// TwinCAT 3 PLC project L2SIVacuum
// Title: LCLS Vacuum
// Company: SLAC - LCLS
// Author: LCLS ECS-Platforms
// ProjectVersion: 2.6.6
// ProgramVersion: 3.1.4026.17
// libraries:
//   LCLS General, * (SLAC)
//   PMPS, * (SLAC - LCLS)
//   Tc2_DataExchange, * (Beckhoff Automation GmbH)
//   Tc2_EtherCAT, * (Beckhoff Automation GmbH)
//   Tc2_ModbusSrv, * (Beckhoff Automation GmbH)
//   Tc2_SerialCom, * (Beckhoff Automation GmbH)
//   Tc2_Standard, * (Beckhoff Automation GmbH)
//   Tc2_System, * (Beckhoff Automation GmbH)
//   Tc2_TcpIp, * (Beckhoff Automation GmbH)
//   Tc2_Utilities, * (Beckhoff Automation GmbH)
//   Tc3_EventLogger, * (Beckhoff Automation GmbH)
//   Tc3_JsonXml, * (Beckhoff Automation GmbH)
//   Tc3_Module, * (Beckhoff Automation GmbH)
//   TcUnit, * (www.tcunit.org)
// project tree:
//   DUTs/Gauges/ E_PressureState.TcDUT, Gauge_Type.TcDUT, ST_VG.TcDUT
//   DUTs/LVDT/ ST_SerLVC4000.TcDUT
//   DUTs/Oerlikon/ ST_TD20Status.TcDUT, ST_TD400Control.TcDUT, ST_TD400Status.TcDUT
//   DUTs/Pfeiffer/ ST_PfeifferControl.TcDUT, ST_PfeifferStatus.TcDUT
//   DUTs/Pumps/ E_PumpState.TcDUT, ST_AgilentPTM.TcDUT, ST_EbaraDryPump.TcDUT, ST_EbaraEVA.TcDUT, ST_EbaraPTM.TcDUT, ST_KashiyamaDryPump.TcDUT, ST_LeyboldPTM.TcDUT, ST_PfeifferPTM.TcDUT, ST_PIP.TcDUT, ST_PTM.TcDUT, ST_RoughPump.TcDUT
//   DUTs/Valves/ E_ValvePositionState.TcDUT, E_VCN.TcDUT, E_2OO3_MODE.TcDUT, E_VGC.TcDUT, ST_ValveBase.TcDUT, ST_VFS.TcDUT, ST_VGC_2S.TcDUT, ST_VRC_NO.TcDUT, ST_VWC_NO.TcDUT, ST_VVC.TcDUT, ST_VCC_NO.TcDUT, ST_VCN.TcDUT, ST_VGC.TcDUT, ST_VRC.TcDUT
//   DUTs/Valves/VAT590/EtherCAT Interface/ E_ControlMode.TcDUT, E_ControlModeSP.TcDUT, E_FatalErrors.TcDUT, ST_ExtendedWarnings.TcDUT, ST_GeneralControlSP.TcDUT, ST_GeneralStatus.TcDUT, ST_GeneralWarnings.TcDUT
//   DUTs/Valves/VAT590/ E_VAT590_AccessMode.TcDUT, E_VAT590_PID_CTRL.TcDUT, E_VCN_VAT590.TcDUT, ST_CoEIndSub.TcDUT, ST_VAT590_COE.TcDUT, ST_VAT590_STATUS.TcDUT, ST_VCN_VAT590.TcDUT
//   GVLs/ Constants.TcGVL, Global_Variables.TcGVL, GVL_MacroSensorsParameters.TcGVL, GVL_PfeifferParameters.TcGVL
//   / PlcTask.TcTTO
//   POUs/ADS/ FB_ADS.TcPOU, FB_ADS_WATCHDOG.TcPOU, FB_TBOOL_ADS.TcPOU
//   POUs/Functions/Deprecated/Gauges/ FB_MKS317A.TcPOU, FB_MKS500_EP.TcPOU, FB_PressureState.TcPOU
//   POUs/Functions/Deprecated/Valves/ FB_VCC.TcPOU, FB_VCC_NO.TcPOU, FB_VGC_AP.TcPOU, FB_VGC_EBD.TcPOU
//   POUs/Functions/Gauges/ FB_901_ECAT.TcPOU, FB_9XX.TcPOU, FB_972.TcPOU, FB_IE514.TcPOU, FB_MX7M.TcPOU, FB_MKS355.TcPOU, FB_GaugeBase.TcPOU, FB_CVM201.TcPOU, FB_CCM501.TcPOU, FB_IMG401.TcPOU, FB_MKS909.TcPOU, FB_MKS909_RBK.TcPOU, FB_CMR362.TcPOU, FB_GCM.TcPOU, FB_ITR90.TcPOU, FB_MKS392.TcPOU, FB_MKS500.TcPOU, FB_MKS722.TcPOU, FB_MKS_937A.TcPOU, FB_MKS317.TcPOU, FB_MKS275.TcPOU, FB_MKS_937B.TcPOU, FB_MKS422.TcPOU
//   POUs/Functions/Gauges/Interfaces/ FB_GaugeModbus.TcPOU, FB_Gauge_Interface.TcPOU, FB_TGCC_ADS.TcPOU, FB_TGPI_ADS.TcPOU, FB_GaugeSelection.TcPOU (not stored)
//   POUs/Functions/Pumps/ FB_EbaraDryPump.TcPOU, FB_EbaraEVA.TcPOU, FB_KashiyamaPump.TcPOU, FB_KashiyamaPump_G.TcPOU, FB_PIP_Gamma.TcPOU, FB_PIP_Gamma_V2.TcPOU, FB_PIP_SIP.TcPOU, FB_PTM_Agilent.TcPOU, FB_PTM_Ebara_011M.TcPOU, FB_PTM_Ebara_010M.TcPOU, FB_PTM_MagDriveDigital.TcPOU, FB_PTM_Pfeiffer.TcPOU, FB_PTM_TurboDrive.TcPOU, FB_PTM_TwisTorr.TcPOU, FB_Pump.TcPOU, FB_ScrollPump.TcPOU
//   POUs/Functions/Pumps/functions/ FB_TurboExtLogic.TcPOU, F_TurboExtILK_NO.TcPOU, F_TurboExtILKLogic.TcPOU, F_TurboExtILKLogic_2.TcPOU, F_TurboExtILK_NO_1.TcPOU
//   POUs/Functions/Pumps/Interfaces/ FB_PIP_Interface_In.TcPOU, FB_PIP_Interface_Out.TcPOU, FB_TPIP_ADS.TcPOU
//   POUs/Functions/Valves/ FB_Kashiyama_VRC.TcPOU, FB_MKS248.TcPOU, FB_TurbVentvalve_NO.TcPOU, FB_Valve.TcPOU, FB_VCN_VAT590.TcPOU, FB_VFS.TcPOU, FB_VFS_2OO3.TcPOU, FB_VGC_2S.TcPOU, FB_VRC_DA.TcPOU, FB_VRC_EBD.TcPOU, FB_VRC_NC_ClsLS.TcPOU, FB_VRC_NO.TcPOU, FB_VRC_NO_FFO.TcPOU, FB_VVC.TcPOU, FB_VCN.TcPOU, FB_VGC.TcPOU, FB_VRC.TcPOU, FB_VRC_OK_CLS.TcPOU
//   POUs/Functions/Valves/functions/ F_RoughPumpInlet_ILK.TcPOU, F_TurboGateValve_ILK.TcPOU, F_TurboGateValve_ILK_1.TcPOU, F_TurboGateValve_Protection_ILK.TcPOU, F_TURBO_VRC_ILK.TcPOU, F_VALVE_REL_ILK.TcPOU, F_VRC_DIODE_ILK_OK.TcPOU, F_VRC_DIODE_ILK.TcPOU
//   POUs/Functions/Valves/Interfaces/ FB_TVGC_2S_ADS.TcPOU, FB_VFS_2OO3Interface.TcPOU, FB_VFS_Interface.TcPOU, FB_TVGC_ADS.TcPOU, FB_Valve_Interface.TcPOU, ITF_Valve.TcIO
//   POUs/Serial drivers/LVDT/MacroSensors/ FB_LVC4000Com.TcPOU, FB_LVC4000SerialDriver.TcPOU, FB_LVC4000Transaction.TcPOU
//   POUs/Serial drivers/Pumps/Oerlikon TD20/ FB_OERLIKON_TD20_COM.TcPOU, FB_OERLIKON_TO_PTM.TcPOU, FB_TD20SerialDriver.TcPOU, FB_TD20Transaction.TcPOU, F_CalcTD20Checksum.TcPOU
//   POUs/Serial drivers/Pumps/Oerlikon TD400/ FB_OERLIKON_TD400_COM.TcPOU, FB_OERLIKON_TD400_TO_PTM.TcPOU, FB_TD400SerialDriver.TcPOU, FB_TD400Transaction.TcPOU, F_CalcTD400Checksum.TcPOU
//   POUs/Serial drivers/Pumps/Pfeiffer/ FB_PfeifferSerialDriver.TcPOU, FB_PfeifferTransaction.TcPOU, FB_PFEIFFER_COM.TcPOU, FB_PFEIFFER_TO_PTM.TcPOU, F_CalcPfeifferCheckSum.TcPOU
//   UnitTests/Functions/ V_TO_INT.TcPOU
//   UnitTests/Gauges/ FB_GCC_Test.TcPOU, FB_GHC_Test.TcPOU, FB_GPI_Test.TcPOU
//   UnitTests/ PRG_Test.TcPOU
//   UnitTests/Pumps/ FB_PIP_Test.TcPOU, FB_PTM_Test.TcPOU
//   UnitTests/Valves/ FB_VGC_Test.TcPOU, FB_VRC_Test.TcPOU
//   Version/ Global_Version.TcGVL
// real-time tasks:
//   TASK TestTask: cycle T#10ms, priority 16, ADS port 350
// variable links:
//   L2SIVacuum/L2SIVacuum Instance <-> L2SIVacuum/L2SIVacuum Instance
//     PlcTask Inputs/PRG_Test.fb_GCC_Test.fb_MKS422.i_iPRESS_R <-> PlcTask Outputs/PRG_Test.fb_GCC_Test.i_iPRESS_R
//     PlcTask Inputs/PRG_Test.fb_GPI_Test.fb_MKS275.i_iPRESS_R <-> PlcTask Outputs/PRG_Test.fb_GPI_Test.i_iPRESS_R
//     PlcTask Inputs/PRG_Test.fb_GPI_Test.fb_MKS317.i_iPRESS_R <-> PlcTask Outputs/PRG_Test.fb_GPI_Test.i_iPRESS_R
//     PlcTask Inputs/PRG_Test.fb_PTM_Test.fb_PTM_Ebara_010M.i_iCurrentMon <-> PlcTask Outputs/PRG_Test.fb_PTM_Test.i_iCurrentMon
//     PlcTask Inputs/PRG_Test.fb_PTM_Test.fb_PTM_Ebara_010M.i_iRawSpeed <-> PlcTask Outputs/PRG_Test.fb_PTM_Test.i_iRawSpeed
//     PlcTask Inputs/PRG_Test.fb_PTM_Test.fb_PTM_Ebara_010M.i_iTempMon <-> PlcTask Outputs/PRG_Test.fb_PTM_Test.i_iTempMon
//     PlcTask Inputs/PRG_Test.fb_PTM_Test.q_iSpeedSet <-> PlcTask Outputs/PRG_Test.fb_PTM_Test.i_diCurSpd

CONFIGURATION L2SIVacuum
    RESOURCE PLC ON TwinCAT3
        TASK PlcTask(INTERVAL := T#10ms, PRIORITY := 16);
        PROGRAM PRG_Test WITH PlcTask : PRG_Test;
    END_RESOURCE
END_CONFIGURATION

// ---- DUTs/Gauges/E_PressureState.TcDUT
TYPE E_PressureState :
(
    // Invalid states
    Off,//	 //gc_GaugeValidState - 1,
    GaugeDisconnected, //gc_GaugeValidState -2,
    OoR, //gc_GaugeValidState -6,
    // Ion gauges
    PressInvalid, //gc_GaugeValidState - 3,
    Starting, //gc_GaugeValidState - 4

    //Valid States (Positive)
    Valid, // gc_GaugeValidState set in "Global Variable Folder: Constants"
    ValidHi, //gc_GaugeValidState + 1,
    ValidLo //gc_GaugeValidState + 2,

) INT;
END_TYPE

// ---- DUTs/Gauges/Gauge_Type.TcDUT
TYPE Gauge_Type: (
PG722B := 0, //Baraton Gauge
IG903 := 1 , //Cold Cathode
PG907 := 2 , //Pirani Gauge
IG909:= 3 , //Hot Cathode
PG925 := 4 ); //MicroPirani Gauge
(* This enumeration should match up with the EDM MUX button on the vacuum gauge expert controls screen *)
END_TYPE

// ---- DUTs/Gauges/ST_VG.TcDUT
TYPE ST_VG :
STRUCT
    /// A general gauge structure is used to make the rest of the interlocking simpler. There are some parameters for cold cathodes that are not used by pirani.
    ///These features aren't disabled, they just aren't used, think child/parent classes.
    ///
    {attribute 'pytmc' := '
    pv: PRESS;
    field: HOPR 1000
    field: LOPR 0
    field: PREC 2
    field: EGU "TORR"
    io: i;
    '}
    rPRESS: REAL;  //This is the human-readable pressure
    {attribute 'pytmc' := '
    pv: AT_VAC;
    io: i;
    field: ZNAM FALSE;
    field: ONAM TRUE;
    '}
    xAT_VAC: BOOL;
    {attribute 'pytmc' := '
    pv: PRESS_OK;
    field: ZNAM OFF;
    field: ONAM ON;
    io: i;
    '}
    xPRESS_OK: BOOL;
    {attribute 'pytmc' := '
    pv: STATE;
    field: ZRST Off;
    field: ONST GaugeDisconnected;
    field: TWST OoR;
    field: THST PressInvalid;
    field: FRST Starting;
    field: FVST Valid;
    field: SXST ValidHi;
    field: SVST ValidLo;
    io: i;
    '}
    eState	:	E_PressureState;
    (* EPICS Controls *)
    {attribute 'pytmc' := '
    pv: HV_SW;
    io: io;
    field: ZNAM OFF;
    field: ONAM ON;
    '}
    xHV_SW: BOOL; // High Voltage Switch from epics
    {attribute 'pytmc' := '
    pv: Auto_On;
    field: ZNAM FALSE;
    field: ONAM TRUE;
    io:io;
    '}
    xAutoOn : BOOL := TRUE;
    {attribute 'pytmc' := '
    pv: AutoOn_timer;
    io:i;
    '}
    iAutoOnTimer : INT;
    /// Controls and I/Os
    {attribute 'pytmc' := '
    pv: PRESS_AI;
    io: i;
    '}
    i_iPRESS_R  :INT; // input Pressure // Link to analog Input
    {attribute 'pytmc' := '
    pv: HV_ON;
    io: i;
    '}
    i_xHV_ON	: BOOL; //  True when High Voltage is on
    {attribute 'pytmc' := '
    pv: DISC_ACTIVE;
    field: ZNAM NO DISC;
    field: ONAM DISC ACTIVE;
    io: i;
    '}
    i_xDisc_Active : BOOL;// Discharge Current Active
    {attribute 'pytmc' := '
    pv: HV_DIS_DO;
    io: i;
    field: ZNAM FALSE ;
    field: ONAM TRUE ;
    '}
    q_xHV_DIS : BOOL; // Enable High Voltage when True
    //
    wHV_RO: WORD;

    /// Bakeout bit
    xBAKEOUT: BOOL;

    //enum for gauge type - will replace iType
    eTYPE: Gauge_Type := PG907;
    //Gauge type, deprecated (default to pirani)
    iTYPE: INT := 2;
    // Index location of the associated Pirani Gauge
    wPG: WORD;


    xTurnOnTime: BOOL;/// Turn on Timers for cold cathode warmup

    iVacSp	:	INT;/// At vacuum setpoint for all gauges
    {attribute 'pytmc' := '
    pv: VAC_SP;
    io:io;
    field: HOPR 1000
    field: LOPR 0
    field: PREC 2
    field: EGU "TORR"
    autosave_pass1: VAL DESC
    '}
    rVAC_SP: REAL := 0.001; /// At vacuum setpoint for all gauges
    /// Protection setpoint for ion gauges at which the gauge turns off, not used for pirani
    {attribute 'pytmc' := '
    pv: PRO_SP;
    io: io;
    field: HOPR 1000
    field: LOPR 0
    field: PREC 2
    field: EGU "TORR"
    autosave_pass1: VAL DESC
    '}
    rPRO_SP: REAL := 0.001;
    {attribute 'pytmc' := '
    pv: SP_HYS;
    io: io;
    field: HOPR 1000
    field: LOPR 0
    field: PREC 2
    field: EGU "TORR"
    autosave_pass1: VAL DESC
    '}
    /// Protection setpoint hysteresis
    rHYS_PR: REAL := 0.001;
    {attribute 'pytmc' := '
    pv: ILK_OK;
    field: ZNAM NOT OK ;
    field: ONAM OK ;
    io: i;
    '}
    xILKOk	:	BOOL; (* also a control *)
    {attribute 'pytmc' := '
    pv: LOGGER;
    io: io;
    field: ZNAM OFF ;
    field: ONAM ON ;
    '}
    xLog : BOOL:=TRUE;
    //Required for other devices using this gauge as interlock
    sPath: STRING;

    /// Full scale pressure in Torr for baratron pressure conversion
    rFULL_SCALE: REAL := 1000;

END_STRUCT
END_TYPE

// ---- DUTs/LVDT/ST_SerLVC4000.TcDUT
TYPE ST_SerLVC4000 :
STRUCT
    (* Readbacks *)
    {attribute 'pytmc' := '
    pv: voltage;
    io: i;
    '}
    i_iOut	:	INT; //Output voltage
    (* Controls *)
    {attribute 'pytmc' := '
    pv: ADC_COEFF;
    io: io;
    '}
    q_rADCsl	:	REAL; //ADC slope coeff
    {attribute 'pytmc' := '
    pv: ADC_OFFSET;
    io: io;
    '}
    q_rADCos	:	REAL; //ADC offset
    {attribute 'pytmc' := '
    pv: CALIB_SET;
    io: io;
    '}
    q_xCal	:	BOOL; //Activate calibration mode
    {attribute 'pytmc' := '
    pv: DISP_SET;
    io: io;
    '}
    q_xFull	:	BOOL; //Set full displacement during calibration
    {attribute 'pytmc' := '
    pv: ZERO_SET;
    io: io;
    '}
    q_xZero	:	BOOL; //Set zero during calibration
    {attribute 'pytmc' := '
    pv: GAIN_SET;
    io: io;
    '}
    q_iGain	:	INT; //Set instrument gain
    {attribute 'pytmc' := '
    pv: CALIB_ABORT;
    io: io;
    '}
    q_xAbortCal	:	BOOL; //Abort calibration mode
    (* Internal params *)
    {attribute 'pytmc' := '
    pv: ADDR;
    io: io;
    '}
    iAddr	:	INT; //RS485 address
    xTimeout	:	BOOL; //Timeout (true if no comm)
END_STRUCT
END_TYPE

// ---- DUTs/Oerlikon/ST_TD20Status.TcDUT
TYPE ST_TD20Status :  (* Serial communication defined in Oerlikon Leybold Manual 17200048 *)
STRUCT
    /// Received Status Word
    wStatusWord: WORD;
    /// Current stator frequency
    {attribute 'pytmc' := '
    pv: Frequency;
    io: i;
    '}
    wFrequency_P3: WORD;
    /// Current intermediate circuit voltage
    {attribute 'pytmc' := '
    pv: Voltage;
    io: i;
    '}
    wVoltage_P4: WORD;
    /// Current motor current
    {attribute 'pytmc' := '
    pv: MotorCurrent;
    io: i;
    '}
    wMotorCurrent_P5: WORD;
    /// Current frequency converter temperature
    {attribute 'pytmc' := '
    pv: Temperature;
    io: i;
    '}
    wConverterTemp_P11: WORD;
    /// Critical frequency
    {attribute 'pytmc' := '
    pv: CriticalFrequency;
    io: i;
    '}
    wCriticalFreq_P20: WORD;
    /// Max. Current Factor
    {attribute 'pytmc' := '
    pv: MaxCurrentFactor;
    io: i;
    '}
    wMaxCurrentFactor_P21: WORD;
    /// Setpoint Frequecy
    {attribute 'pytmc' := '
    pv: SetPointFreq;
    io: i;
    '}
    wSetpointFreq_P24: WORD;
    /// Max. run up time
    {attribute 'pytmc' := '
    pv: MaxRunUpTime;
    io: i;
    '}
    wMaxRunUpTime_P32: WORD;
    /// Current pump temperature
    {attribute 'pytmc' := '
    pv: PumpTemp;
    io: i;
    '}
    wPumpTemp_P127: WORD;
    /// most recent error code
    {attribute 'pytmc' := '
    pv: ErrorCode;
    io: i;
    '}
    wErrorCode_P171: WORD;
END_STRUCT
END_TYPE

// ---- DUTs/Oerlikon/ST_TD400Control.TcDUT
TYPE ST_TD400Control :  (* Serial communication defined in Oerlikon Leybold Manual GA05281_002_C0 *)
STRUCT
    {attribute 'pytmc' := '
    pv: SetPumpSpeed;
    io: i;
    '}
    wSetSetpointFreq_P24: WORD; // speed setting in Hz
END_STRUCT
END_TYPE

// ---- DUTs/Oerlikon/ST_TD400Status.TcDUT
TYPE ST_TD400Status :  (* Serial communication defined in Oerlikon Leybold Manual 17200048 *)
STRUCT
    /// Received Status Word
    wStatusWord: WORD;
    /// Current stator frequency
    {attribute 'pytmc' := '
    pv: Frequency;
    io: i;
    '}
    wFrequency_P3: WORD;
    /// Current intermediate circuit voltage
    {attribute 'pytmc' := '
    pv: Voltage;
    io: i;
    '}
    wVoltage_P4: WORD;
    /// Current motor current
    {attribute 'pytmc' := '
    pv: MotorCurrent;
    io: i;
    '}
    wMotorCurrent_P5: WORD;
    /// Current frequency converter temperature
    {attribute 'pytmc' := '
    pv: Temperature;
    io: i;
    '}
    wConverterTemp_P11: WORD;
    /// Maximum setpoint frequency
    {attribute 'pytmc' := '
    pv: MaxSetpoinFreq;
    io: i;
    '}
    wMaxSetpointFreq_P18: WORD;
    /// Minimum setpoint frequency
    {attribute 'pytmc' := '
    pv: MinSetpoinFreq;
    io: i;
    '}
    wMinSetpointFreq_P19: WORD;
    /// Critical frequency
    {attribute 'pytmc' := '
    pv: CriticalFrequency;
    io: i;
    '}
    wCriticalFreq_P20: WORD;
    /// Setpoint Frequecy
    {attribute 'pytmc' := '
    pv: SetPointFreq;
    io: i;
    '}
    wSetpointFreq_P24: WORD;
    /// Max. run up time
    {attribute 'pytmc' := '
    pv: MaxRunUpTime;
    io: i;
    '}
    wMaxRunUpTime_P32: WORD;
    /// Current pump temperature
    {attribute 'pytmc' := '
    pv: PumpTemp;
    io: i;
    '}
    wPumpTemp_P127: WORD;
    /// most recent error code
    {attribute 'pytmc' := '
    pv: ErrorCode;
    io: i;
    '}
    wErrorCode_P171: WORD;
END_STRUCT
END_TYPE

// ---- DUTs/Pfeiffer/ST_PfeifferControl.TcDUT
TYPE ST_PfeifferControl :
STRUCT
    /// enables communication
    {attribute 'pytmc' := '
    pv: COMM_EN;
    io: io;
    '}
    xEnableComm: BOOL;
    /// RS-485 Address
    {attribute 'pytmc' := '
    pv: ADDR;
    io: io;
    '}
    iSerialAddress: INT;
    {attribute 'pytmc' := '
    pv: EXT_ILK_OK;
    field: ZNAM ILK ACTIVE;
    field: ONAM ILK OK;
    io: i;
    '}
    /// pumping station (equivalent to ilk bit for varian)
    xPumpingStation_010: BOOL;
    {attribute 'pytmc' := '
    pv: SetPumpSpeed;
    io: i;
    '}
    iSetRotationSpeed_707: INT :=100; /// speed setting in % (normally 100%)
    /// RUN_DO bit
    {attribute 'pytmc' := '
    pv: RUN_DO;
    io: i;
    '}
    xMotorPump_023: BOOL;
    {attribute 'pytmc' := '
    pv: GAS_MODE;
    io: io;
    '}
    iGasMode_027: INT;
    /// interlock bit
     {attribute 'pytmc' := '
    pv: ILK_OK;
    field: ZNAM ILK ACTIVE;
    field: ONAM ILK OK;
    io: i;
    '}
    xIlk: BOOL;
    /// run/start bit
    {attribute 'pytmc' := '
    pv: RUN_SW;
    io: io;
    '}
    xRunSW: BOOL;
    /// error acknowledgement/reset bit
    {attribute 'pytmc' := '
    pv: ERR_RST;
    io: io;
    '}
    xErrorAck_009: BOOL;
    /// power consumption setting in % (normally 100%)
    uiPowerPct_708: UINT;
    xSetSpdMode_026: BOOL;
END_STRUCT
END_TYPE

// ---- DUTs/Pfeiffer/ST_PfeifferStatus.TcDUT
TYPE ST_PfeifferStatus :
STRUCT
    {attribute 'pytmc' := '
    pv: PumpingStation_RBV;
    field: ZNAM ILK ACTIVE;
    field: ONAM ILK OK;
    io: i;
    '}
    xPumpingStation_010: BOOL;
    {attribute 'pytmc' := '
    pv: PumpingStation_RBV;
    field: ZNAM FALSE;
    field: ONAM TRUE;
    io: i;
    '}
    xMotorPump_023: BOOL;
    {attribute 'pytmc' := '
    pv: GasMode_RBV;
    io: i;
    '}
    iGasMode_027: INT;
    {attribute 'pytmc' := '
    pv: ErrorMessage_RBV;
    io: i;
    '}
    sErrorCode_303: STRING;
    {attribute 'pytmc' := '
    pv: ErrorCode_RBV;
    io: i;
    '}
    iErrorCode_303	:	INT;
    {attribute 'pytmc' := '
    pv: WarningCode_RBV;
    io: i;
    '}
    iWarningCode_303	:	INT;
    {attribute 'pytmc' := '
    pv: ExcessPumpTemp_RBV;
    field: ZNAM FALSE;
    field: ONAM TRUE;
    io: i;
    '}
    xExcessTempPump_305: BOOL;
    {attribute 'pytmc' := '
    pv: TotationSpeedAttn_RBV;
    field: ZNAM FALSE;
    field: ONAM TRUE;
    io: i;
    '}
    xRotationSpeedAttn_306: BOOL;
    {attribute 'pytmc' := '
    pv: PumpAccelerating_RBV;
    field: ZNAM FALSE;
    field: ONAM TRUE;
    io: i;
    '}
    xPumpAccelerating_307: BOOL;
    {attribute 'pytmc' := '
    pv: PumpSpeed_RBV;
    io: i;
    '}
    diActiveRotationSpeed_309: DINT;
    {attribute 'pytmc' := '
    pv: DriveCurrent_RBV;
    io: i;
    '}
    lrDriveCurrent_310: LREAL;
    {attribute 'pytmc' := '
    pv: DrivePower_RBV;
    io: i;
    '}
    diDrivePower_316: DINT;
    {attribute 'pytmc' := '
    pv: TempElect_RBV;
    io: i;
    '}
    diTempElec_326: DINT;
    {attribute 'pytmc' := '
    pv: TempPump_RBV;
    io: i;
    '}
    diTempPmpBot_330: DINT;
    {attribute 'pytmc' := '
    pv: TempBearing_RBV;
    io: i;
    '}
    diTempBearng_342: DINT;
    {attribute 'pytmc' := '
    pv: TempMotor_RBV;
    io: i;
    '}
    diTempMotor_346: DINT;
    {attribute 'pytmc' := '
    pv: Power_RBV;
    io: i;
    '}
    uiPowerPct_708: UINT;
    {attribute 'pytmc' := '
    pv: Timeout_RBV;
    field: ZNAM FALSE;
    field: ONAM TRUE;
    io: i;
    '}
    xTimeout: BOOL;
    iSetRotationSpeed_707 : INT;
    iSetSpdMode_026: INT;
    xErrorAcknowledged: BOOL; //Not actually read back from the pump, but tells us ErrAck has processed
END_STRUCT
END_TYPE

// ---- DUTs/Pumps/E_PumpState.TcDUT
TYPE E_PumpState :
(
pumpSTOPPED	:= 0,
pumpSTARTING	:= 1,
pumpRUNNING	:= 2,
pumpFAULT := 3,
pumpSTOPPING :=4
);
END_TYPE

// ---- DUTs/Pumps/ST_AgilentPTM.TcDUT
TYPE ST_AgilentPTM EXTENDS ST_PTM :
STRUCT

(* Inputs *)
    (* 24V in Ramp state; 0V for others *)
    {attribute 'pytmc' := '
    pv: START;
    field: ZNAM FALSE;
    field: ONAM TRUE;
    io: i;
    '}
    i_xSTART :	BOOL;

    (* setpoint related to frequency *)
    {attribute 'pytmc' := '
    pv: R1Status;
    field: ZNAM FALSE;
    field: ONAM AT SPEED;
    io: i;
    '}
    i_xR1	:  BOOL;

    (* setpoint related to Power *)
    {attribute 'pytmc' := '
    pv: R2Status;
    field: ZNAM FALSE;
    field: ONAM TRUE;
    io: i;
    '}
    i_xR2	:  BOOL;

    (* low speed mode *)
    {attribute 'pytmc' := '
    pv: LSPD;
    field: ZNAM FALSE;
    field: ONAM TRUE;
    io: i;
    '}
    i_xLSpd	:  BOOL;


    (* Fault input*)
    //i_xFault : BOOL;  Inherit ST_PTM.xFault



(* controls *)
    (* Start/Stop -
        q_RunDo ;   Inherit ST_PTM.
     *)

    (* Low speed control *)
    {attribute 'pytmc' := '
    pv: LSPD_DO;
    field: ZNAM FALSE;
    field: ONAM TRUE;
    io: i;
    '}
    q_xLSpd		:  BOOL;

    (*Soft start *)
    {attribute 'pytmc' := '
    pv: XSS_DO;
    field: ZNAM FALSE;
    field: ONAM TRUE;
    io: i;
    '}
    q_xSS   	:  BOOL;

    (*pump Lock*)
    {attribute 'pytmc' := '
    pv: FaultLock;
    field: ZNAM FALSE;
    field: ONAM TRUE;
    io: i;
    '}
    xPumpFaultLock : BOOL := FALSE;
    // i_xPumpLockReset: BOOL := FALSE; Inherit ST_PTM.xReset
    // Error messages
    {attribute 'pytmc' := '
    pv: ErrorMessage;
    io: i;
    '}
    sError : STRING;
    {attribute 'pytmc' := '
    pv: Power_MON;
    io: i;
    field: PREC 2
    field: EGU "W";
    '}
    i_rPowerMon : REAL;

END_STRUCT
END_TYPE

// ---- DUTs/Pumps/ST_EbaraDryPump.TcDUT
TYPE ST_EbaraDryPump EXTENDS ST_RoughPump :
STRUCT
(* Extension of the rough pump archetype for ebara
Applicable to:
EV-S20
EV-S50
EV-S100
EV-S200
*)

//Controls
{attribute 'pytmc' := '
    pv: MPStart;
    field: ZNAM FALSE;
    field: ONAM TRUE;
    io: i;
    '}
q_xMPStart	:	BOOL; //Main Pump start
{attribute 'pytmc' := '
    pv: BPStart;
    field: ZNAM FALSE;
    field: ONAM TRUE;
    io: i;
    '}
q_xBPStart	:	BOOL; // Booster Pump start (this can be started by the pump automatically)

xBPIlk	:	BOOL;	//Booster pump interlock
rBPIlkSP	:	REAL := 30; //Booster pump pressure setpoint
tonBP	:	TON := (PT:=T#5S); //Timer for pressure and valve stability


//Readbacks
{attribute 'pytmc' := '
    pv: MPStatus;
    field: ZNAM FALSE;
    field: ONAM TRUE;
    io: i;
    '}
i_xMPStatus	:	BOOL; //MP status
{attribute 'pytmc' := '
    pv: BPStatus;
    field: ZNAM FALSE;
    field: ONAM TRUE;
    io: i;
    '}
i_xBPStatus	:	BOOL; //BP status
{attribute 'pytmc' := '
    pv: WARN_DI;
    field: ZNAM FALSE;
    field: ONAM TRUE;
    io: i;
    '}
i_xWarning	:	BOOL; //Warning status
{attribute 'pytmc' := '
    pv: ALARM;
    field: ZNAM FALSE;
    field: ONAM TRUE;
    io: i;
    '}
i_xAlarm	:	BOOL; //Alarm, maps to error
{attribute 'pytmc' := '
    pv: REMOTE;
    field: ZNAM FALSE;
    field: ONAM TRUE;
    io: i;
    '}
i_xRemote	:	BOOL; //Remote control status


END_STRUCT
END_TYPE

// ---- DUTs/Pumps/ST_EbaraEVA.TcDUT
TYPE ST_EbaraEVA EXTENDS ST_RoughPump:
STRUCT

(* Output *)
    //q_xRunDO 	:	BOOL; in Rough PUMP


(* Input *)
{attribute 'pytmc' := '
    pv: REMOTE;
    field: ZNAM FALSE;
    field: ONAM TRUE;
    io: io;
    '}
    q_xRemote	:	BOOL;
    {attribute 'pytmc' := '
    pv: ALARM_OK;
    field: ZNAM FALSE;
    field: ONAM TRUE;
    io: i
    '}
    i_xAlarmOK	:	BOOL;

    {attribute 'pytmc' := '
    pv: RUN_DI;
    field: ZNAM FALSE;
    field: ONAM TRUE;
    io: i
    '}
    i_xIsRun		:	BOOL;


    {attribute 'pytmc' := '
    pv: RST_SW;
    field: ZNAM FALSE;
    field: ONAM TRUE;
    io: io;
    '}
    q_xReset	:	BOOL; //For resetting faults


END_STRUCT
END_TYPE

// ---- DUTs/Pumps/ST_EbaraPTM.TcDUT
TYPE ST_EbaraPTM EXTENDS ST_PTM :
STRUCT
(* Extension of the PTM archetype for Ebara turbo controllers
Applicable to:
ETC series
*)
//Controls
    {attribute 'pytmc' := '
    pv: START;
    field: ZNAM FALSE;
    field: ONAM TRUE;
    io: i;
    '}
q_xStart   : BOOL; //Outputs - FB decides if these are actually set
    {attribute 'pytmc' := '
    pv: STOP;
    field: ZNAM FALSE;
    field: ONAM TRUE;
    io: i;
    '}
q_xStop    : BOOL;
    {attribute 'pytmc' := '
    pv: RESET;
    field: ZNAM FALSE;
    field: ONAM TRUE;
    io: i;
    '}
q_xReset   : BOOL; // xReset is momentary reset switch - resets protection functions
    {attribute 'pytmc' := '
    pv: PROT;
    field: ZNAM FALSE;
    field: ONAM TRUE;
    io: i;
    '}
q_xProtection : BOOL; //NC. If opened, pump will decelerate/not start
    {attribute 'pytmc' := '
    pv: SETSPEED
    field: ZNAM FALSE;
    field: ONAM TRUE;
    io: io
    '}
iq_xSpeedSet    : BOOL; //Request to set speed
    {attribute 'pytmc' := '
    pv: SPEED_REQ
    io: io
    field: EGU "Hz"
    '}
q_iSpeedSet   : DINT; //Requested speed (min. 100Hz)
    {attribute 'pytmc' := '
    pv: OVRD_ON
    field: ZNAM OFF;
    field: ONAM ON;
    io: io
    '}
i_xOverride   : BOOL; //Override mode - ignores interlocks

//Readbacks - also has Accel/At speed/Decel/Fault/Cur Speed (min 100RPM)
    {attribute 'pytmc' := '
    pv: ROTATE_STATUS
    field: ZNAM FALSE;
    field: ONAM ROTATING;
    io: i
    '}
i_xRotate : BOOL; //If open, pump is rotating
    {attribute 'pytmc' := '
    pv: DECEL
    field: ZNAM FALSE;
    field: ONAM DECELERATING;
    io: i
    '}
i_xDecel  : BOOL; //If closed, brake engaged (pump decelerating)
    {attribute 'pytmc' := '
    pv: FAULT_OK
    field: ZNAM FALSE;
    field: ONAM TRUE;
    io: i
    '}
i_xNCFault  : BOOL; //Normally closed fault wiring. If false, there is a fault, or cable is unplugged.



END_STRUCT
END_TYPE

// ---- DUTs/Pumps/ST_KashiyamaDryPump.TcDUT
TYPE ST_KashiyamaDryPump EXTENDS ST_RoughPump:
STRUCT

(* Output *)
    //q_xRunDO 	:	BOOL; in Rough PUMP
    {attribute 'pytmc' := '
    pv: RESET_DO;
    field: ZNAM FALSE;
    field: ONAM TRUE;
    io: i
    '}
    q_xResetDo	: 	BOOL;
    {attribute 'pytmc' := '
    pv: LSPD_DO;
    field: ZNAM FALSE;
    field: ONAM TRUE;
    io: i
    '}
    q_xLspdDo	: 	BOOL;
	{attribute 'pytmc' := '
    pv: REMOTE_ENBL;
    field: ZNAM FALSE;
    field: ONAM TRUE;
    io: i
    '}
    q_xRemoteEn	: 	BOOL;
	


(* Input *)
{attribute 'pytmc' := '
    pv: REMOTE;
    field: ZNAM FALSE;
    field: ONAM TRUE;
    io: i
    '}
    i_xRemote	:	BOOL;

    {attribute 'pytmc' := '
    pv: ALARM_OK;
    field: ZNAM FALSE;
    field: ONAM TRUE;
    io: i
    '}
    i_xAlarmOK	:	BOOL;
    {attribute 'pytmc' := '
    pv: WARN_OK;
    field: ZNAM FALSE;
    field: ONAM TRUE;
    io: i
    '}
    i_xWarningOK	:	BOOL;
    {attribute 'pytmc' := '
    pv: RUN_DI;
    field: ZNAM FALSE;
    field: ONAM TRUE;
    io: i
    '}
    i_xIsRun		:	BOOL;

(* Logic status *)

    xLspd_IlkENA:   BOOL;

(* EPICS *)
    //xRunSW		:	BOOL; in Rough PUMP
    {attribute 'pytmc' := '
    pv: RESET_SW;
    field: ZNAM FALSE;
    field: ONAM TRUE;
    io: io
    '}
    xResetSW	:	BOOL; //For resetting faults
    {attribute 'pytmc' := '
    pv: LSPD_SW;
    field: ZNAM FALSE;
    field: ONAM TRUE;
    io: io
    '}
    xLspdSW     :   BOOL;
    LowSP  :   REAL := 0.02; //Torr
    HighSP :   REAL; //Torr
    RdyTmr : REAL;
END_STRUCT
END_TYPE

// ---- DUTs/Pumps/ST_LeyboldPTM.TcDUT
TYPE ST_LeyboldPTM EXTENDS ST_PTM :
STRUCT
(* Extension of the PTM archetype for Oerlikon turbo controllers
Applicable to:
Mag Drive Digital
Mag Drive S
More?
*)
//Readbacks
    {attribute 'pytmc' := '
    pv: DECEL;
    field: ZNAM FALSE;
    field: ONAM TRUE;
    io: i;
    '}
    i_xDecel	:	BOOL;
    {attribute 'pytmc' := '
    pv: PWR_RBV;
    io: i;
    '}
    i_diPwr   	:   DINT;
    i_diElecTemp:	DINT;
    {attribute 'pytmc' := '
    pv: OVR_TEMP;
    field: ZNAM FALSE;
    field: ONAM TRUE;
    io: i;
    '}
    i_xTempFault:	BOOL;
    i_xNCError	:	BOOL; //Using normally closed wiring

//Controls
    {attribute 'pytmc' := '
    pv: REMOTE;
    field: ZNAM FALSE;
    field: ONAM TRUE;
    io: io;
    '}
    q_xRemote :BOOL;
    i_xRemote : BOOL; (* Remote control enabled *)
END_STRUCT
END_TYPE

// ---- DUTs/Pumps/ST_PfeifferPTM.TcDUT
TYPE ST_PfeifferPTM EXTENDS ST_PTM :
STRUCT
(* Extension of the PTM archetype for Pfeiffer turbos
Applicable to:
HiPace series w/ onboard controllers
More?
*)
    {attribute 'pytmc' := '
    pv: RESET;
    field: ZNAM FALSE;
    field: ONAM TRUE;
    io: i;
    '}
    q_xReset   : BOOL;
    //Readbacks
    {attribute 'pytmc' := '
    pv: PWR_RBV;
    io: i;
    '}
    i_diPwr		:	DINT;
    {attribute 'pytmc' := '
    pv: TempElec_RBV;
    io: i;
    '}
    i_diElecTemp	:	DINT;
    {attribute 'pytmc' := '
    pv: TempPump_RBV;
    io: i;
    '}
    i_diBtmTemp:	DINT;
    {attribute 'pytmc' := '
    pv: TempBearing_RBV;
    io: i;
    '}
    i_diBrngTemp:	DINT;
    {attribute 'pytmc' := '
    pv: TempMotor_RBV;
    io: i;
    '}
    i_diMtrTemp:	DINT;
    {attribute 'pytmc' := '
    pv: ErrorCode_RBV;
    io: i;
    '}
    i_iErrorCode	:	INT; //might change these to enumeration someday
    {attribute 'pytmc' := '
    pv: WarningCode_RBV;
    io: i;
    '}
    i_iWarningCode	:	INT;
    {attribute 'pytmc' := '
    pv: TempFault_RBV;
    field: ZNAM FALSE;
    field: ONAM TRUE;
    io: i;
    '}
    i_xTempFault	:	BOOL;
    {attribute 'pytmc' := '
    pv: Power_RBV;
    io: i;
    '}
    i_uiPowerPctRbk :   UINT;

    {attribute 'pytmc' := '
    pv: SET_SPEED;
    io: io;
    field: EGU "Hz"
    '}
    i_dSetSpd	:	DINT;

    {attribute 'pytmc' := '
    pv: SET_SPEED_MODE;
    io: io;
    field: ZNAM FALSE;
    field: ONAM TRUE;
    '}
    q_bSetSpd	:	BOOL;

//Controls
    q_uiPowerPct : UINT := 100; //Should normally be 100

END_STRUCT
END_TYPE

// ---- DUTs/Pumps/ST_PIP.TcDUT
TYPE ST_PIP :
STRUCT
(* Read back *)
// 	i_xHVisON : BOOL;

(* Interlock *)
    {attribute 'pytmc' := '
    pv: ILK_OK;
    field: ZNAM NOT OK ;
    field: ONAM OK ;
    io: i;
    '}
       xILKOk : BOOL;

    {attribute 'pytmc' := '
    pv: ERROR;
    field: ZNAM FALSE ;
    field: ONAM TRUE ;
    io: i;
    '}
       xError : BOOL;

    {attribute 'pytmc' := '
    pv: AT_VAC_SP;
    io: io;
    field: HOPR 1000
    field: LOPR 0
    field: PREC 2
    field: EGU "TORR"
    autosave_pass1: VAL DESC
    '}
    rHVEna_SP : REAL := 1.0E-4;

    {attribute 'pytmc' := '
    pv: ILK_DEVICE;
    io: i;
    '}
    sIlkDeviceName: STRING;
    //Required for other devices using this gauge as interlock
    sPath: STRING;

(* EPICS Controls *)
    {attribute 'pytmc' := '
    pv: HV_SW;
    io: io;
    field: ZNAM OFF;
    field: ONAM ON;
    '}
    xHVEna_SW : BOOL;
    {attribute 'pytmc' := '
    pv: Auto_On;
    field: ZNAM FALSE;
    field: ONAM TRUE;
    io:io;
    '}
    xAutoOn : BOOL:=TRUE;

    {attribute 'pytmc' := '
    pv: AutoOn_timer;
    io:i;
    '}
    iAutoOnTimer : INT;

    {attribute 'pytmc' := '
    pv: OVRD_ON ;
    field: ZNAM Override OFF ;
    field: ONAM Override ON;
    io: io;
    '}
    xOverrideMode	:	BOOL; (* Shows the override status of this valve *)

    {attribute 'pytmc' := '
    pv: FORCE_START;
    io: io;
    field: ZNAM FALSE;
    field: ONAM FORCE START;
    '}
    pv_xOvrdStart	:	BOOL;


    {attribute 'pytmc' := '
    pv: SP_HYS;
    io: io;
    field: HOPR 1000
    field: LOPR 0
    field: PREC 2
    field: EGU "TORR"
    autosave_pass1: VAL DESC
    '}
    /// Protection setpoint hysteresis
    rHYS_PR: REAL := 0.001;
    {attribute 'pytmc' := '
    pv: AI_Offset;
    io: io;
    '}
    iOffset: INT:=13;
    {attribute 'pytmc' := '
    pv: Inverted;
    field: ZNAM NORMAL;
    field: ONAM INVERTED;
    io: io;
    '}
    bOutputInverted : BOOL;
(* IO Controls *)
    {attribute 'pytmc' := '
    pv: HV_DO;
    field: ZNAM OFF;
    field: ONAM ON;
    io: i;
    '}
    q_xHVEna_DO : BOOL;	// Enable High Voltage when True // 'TcLinkTo' (EL1124) ^Input
    {attribute 'pytmc' := '
    pv: PRESS;
    field: HOPR 1000
    field: LOPR 0
    field: PREC 2
    field: EGU "TORR"
    io: i;
    '}
    rPRESS: REAL;  //
    {attribute 'pytmc' := '
    pv: PRESS_AI;
    io: i;
    '}
    i_iPRESS: REAL;  //
    {attribute 'pytmc' := '
    pv: HV_DI;
    field: ZNAM FALSE;
    field: ONAM TRUE;
    io:i;
    '}
    i_xHV_DI : BOOL; // NO contact // 'TcLinkTo' (EL1004) ^Input

    {attribute 'pytmc' := '
    pv: STATE;
    field: ZRST STOPPED;
    field: ONST STARTING;
    field: TWST RUNNING;
    field: THST FAULT;
    field: FRST STOPPING;
    io: i;
    '}

    eState	:	E_PumpState;

    {attribute 'pytmc' := '
    pv: LOGGER;
    io: io;
    field: ZNAM OFF ;
    field: ONAM ON ;
    '}
    xLog : BOOL:=TRUE;
END_STRUCT
END_TYPE

// ---- DUTs/Pumps/ST_PTM.TcDUT
TYPE ST_PTM :
STRUCT
(* General PTM Structure
Each PTM might have a serial control structure, but all will have a general supervisory control structure

NOTE: This is an archetype, use an extension of this structure for a specific pump (or make one).

*)

(* Controls *)
    {attribute 'pytmc' := '
    pv: RUN_SW;
    field: ZNAM STOP;
    field: ONAM RUN;
    io: io;
    '}
    xRunSW	:	BOOL;
    {attribute 'pytmc' := '
    pv: RST_SW;
    field: ZNAM FALSE;
    field: ONAM TRUE;
    io: io;
    '}
    xResetSW	:	BOOL; //For resetting faults
    {attribute 'pytmc' := '
    pv: RUN_DO;
    io: i;
    '}
    q_RunDO 	:	BOOL;

(* Readbacks *)
    {attribute 'pytmc' := '
    pv: ILK_OK;
    field: ZNAM ILK ACTIVE;
    field: ONAM ILK OK;
    io: i;
    '}
    xExtRunOk	:	BOOL; (* also a control *)
    {attribute 'pytmc' := '
    pv: ACCEL;
    field: ZNAM FALSE;
    field: ONAM TRUE;
    io: i;
    '}
    i_xAccel	:	BOOL;
    {attribute 'pytmc' := '
    pv: AT_SPD;
    field: ZNAM FALSE;
    field: ONAM AT SPEED;
    io: i;
    '}
    i_xAtSpd	:	BOOL;
    {attribute 'pytmc' := '
    pv: SPEED;
    io: i;
    field: EGU "Hz"
    '}
    i_diCurSpd	:	DINT;

    xCommTimeout	:	BOOL := TRUE;  (* Initialized true since we haven't talked to pump yet *)
(* Alarm Outputs *)
    {attribute 'pytmc' := '
    pv: FAULT;
    field: ZNAM FALSE;
    field: ONAM TRUE;
    io: i;
    '}
    i_xFault		:	BOOL; (*FAULT*)
    {attribute 'pytmc' := '
    pv: WARN;
    field: ZNAM FALSE;
    field: ONAM TRUE;
    io: i;
    '}
    i_xWarn		:	BOOL; (* warning *)
    {attribute 'pytmc' := '
    pv: ALARM;
    field: ZNAM FALSE;
    field: ONAM TRUE;
    io: i;
    '}
    i_xALARM	:	BOOL; (* ALARM *)

(* IWS instructions *)
    xActive	:	BOOL; // this bit is set to add the pump to the system
    iPumpGrp 	:	INT; // all members of a pump group start at the same time

(* Operational Setpoints *)
    rForelineSP	:	REAL := 0.5;

    {attribute 'pytmc' := '
    pv: BP_SP;
    io: io;
    field: HOPR 1000
    field: LOPR 0
    field: PREC 2
    field: EGU "TORR"
    autosave_pass1: VAL DESC
    '}
    rBackingPressureSP : REAL := 0.01;
    {attribute 'pytmc' := '
    pv: IP_SP;
    io: io;
    field: HOPR 1000
    field: LOPR 0
    field: PREC 2
    field: EGU "TORR"
    autosave_pass1: VAL DESC
    '}
    rInletPressureSP : REAL := 0.02; //20mTorr
(*State*)
    {attribute 'pytmc' := '
    pv: STATE;
    field: ZRST STOPPED;
    field: ONST STARTING;
    field: TWST RUNNING;
    field: THST FAULT;
    field: FRST STOPPING;
    io: i;
    '}

    eState	:	E_PumpState;

    {attribute 'pytmc' := '
    pv: CURR_MON;
    io: i;
    field: PREC 2
    field: EGU "A";
    '}
    i_rCurrentMon : REAL;

    {attribute 'pytmc' := '
    pv: TEMP_MON;
    io: i;
    field: PREC 2;
    field: EGU "C";
    '}
    i_rTempMon	:	REAL;

    {attribute 'pytmc' := '
    pv: LOGGER;
    io: i;
    field: ZNAM OFF ;
    field: ONAM ON ;
    '}
    xLog : BOOL:=TRUE;


END_STRUCT
END_TYPE

// ---- DUTs/Pumps/ST_RoughPump.TcDUT
TYPE ST_RoughPump :
STRUCT

(* Generic roughing pump controls

NOTE: This is an archetype, use an extension of this structure for a specific pump (or make one).

*)

//Controls
{attribute 'pytmc' := '
    pv: RUN_SW;
    field: ZNAM Stop;
    field: ONAM Start;
    io: io;
    '}
pv_xRunSW	:	BOOL; //epics/ software control switch
{attribute 'pytmc' := '
    pv: RUN_DO;
    field: ZNAM FALSE;
    field: ONAM TRUE;
    io: i
    '}
q_xRunDo 	:   BOOL;

//Status and Readback
{attribute 'pytmc' := '
    pv: ILK_OK;
    field: ZNAM NOT OK ;
    field: ONAM OK ;
    io: i
    '}
xIlkOK	:	BOOL; //Interlock bit, true means OK to run
xExtIlk	:	BOOL; //External interlock, this is where the logic goes
{attribute 'pytmc' := '
    pv: AT_SPD;
    field: ZNAM FALSE;
    field: ONAM TRUE;
    io: i
    '}
xAtSpd	:	BOOL; //Pump at speed setpoint
{attribute 'pytmc' := '
    pv: WARN;
    field: ZNAM FALSE;
    field: ONAM TRUE;
    io: i
    '}
xWrn	:	BOOL; //Pump warning
iWrn	:	BOOL; //Warning state/code
{attribute 'pytmc' := '
    pv: ERROR;
    field: ZNAM FALSE;
    field: ONAM TRUE;
    io: i
    '}
xErr	:	BOOL; //Error summary
iErr	:	BOOL; //Error state/code

(*State*)
    {attribute 'pytmc' := '
    pv: STATE;
    field: ZRST STOPPED;
    field: ONST STARTING;
    field: TWST RUNNING;
    field: THST FAULT;
    field: FRST STOPPING;
    io: i;
    '}

    eState	:	E_PumpState;

END_STRUCT
END_TYPE

// ---- DUTs/Valves/E_ValvePositionState.TcDUT
TYPE E_ValvePositionState :
    (
OPEN	:= 0,
CLOSED	:= 1,
MOVING	:= 2,
INVALID :=3,
OPEN_F :=4
);
END_TYPE

// ---- DUTs/Valves/E_VCN.TcDUT
TYPE E_VCN :
    (
CloseValve	:= 0,
OpenValve	:= 1,
PressureControl	:= 2,
ManualControl	:= 3

    );
END_TYPE

// ---- DUTs/Valves/E_2OO3_MODE.TcDUT
TYPE E_2OO3_MODE :
(
    MODE_2OO3 := 0,
    IG1 := 1,
    IG2 := 2,
    IG3 := 3
);
END_TYPE

// ---- DUTs/Valves/E_VGC.TcDUT
TYPE E_VGC :
(

    Vented,
    AtVacuum,
    ERR_DiffPress,
    ERR_LostVac,
    ERR_ExtFault,
    At_Vac,
    Triggered,
    Vac_Fault,
    Cls_Timeout,
    Opn_Timeout


);
END_TYPE

// ---- DUTs/Valves/ST_ValveBase.TcDUT
TYPE ST_ValveBase :
STRUCT
    (* EPICS Controls *)
    {attribute 'pytmc' := '
    pv: OPN_SW;
    field: ZNAM CLOSE;
    field: ONAM OPEN;
    io: io ;
    '}
    pv_xOPN_SW	: BOOL;
    {attribute 'pytmc' := '
    pv: ALM_RST;
    io: io;
    '}
    pv_xAlmRst	: BOOL;
    {attribute 'pytmc' := '
    pv: FORCE_OPN;
    io: io;
    field: ZNAM FALSE;
    field: ONAM FORCE OPEN;
    '}
    pv_xOvrdOpn	:	BOOL;

    {attribute 'pytmc' := '
    pv: OVRD_ON ;
    field: ZNAM Override OFF ;
    field: ONAM Override ON;
    io: io;
    '}
    xOverrideMode	:	BOOL; (* Shows the override status of this valve *)

(* I/Os*)
(* Readbacks *)
    {attribute 'pytmc' := '
    pv: OPN_DI;
    io: i;
    field: ZNAM FALSE;
    field: ONAM OPEN;
    '}
    i_xOpnLS	: BOOL;
    {attribute 'pytmc' := '
    pv: CLS_DI;
    io: i;
    field: ZNAM FALSE;
    field: ONAM CLOSE;
    '}
    i_xClsLS	: BOOL;
(* Controls *)
    {attribute 'pytmc' := '
    pv: OPN_DO;
    io: i;
    field: ZNAM FALSE;
    field: ONAM TRUE;
    '}
    q_xOPN_DO	: BOOL;
(* Interlocks *)
    {attribute 'pytmc' := '
    pv: EXT_ILK_OK ;
    field: ZNAM NOT OK ;
    field: ONAM OK ;
    io: i ;
    '}
    xEXT_OK	:	BOOL := FALSE;	(* External interlock for custom interlocking in addition to regular DP ilk, this must be set true, or the interlock condition before calling the FB_VGC *)


    {attribute 'pytmc' := '
    pv: OPN_OK;
    field: ZNAM OPN ILK NOT OK ;
    field: ONAM OPN ILK OK ;
    io: i;
     '}
    xOPN_OK	:	BOOL;	(* Final SUM of DP_OK and EXT_OK, needed because it allows the DP ilk to be switched off, see FB_VGC.Dis_DPIlk *)

(* States *)
{attribute 'pytmc' := '
    pv: POS_STATE;
    type: mbbi ;
    field: ZRST OPEN ;
    field: ONST CLOSED ;
    field: TWST MOVING ;
    field: THST INVALID ;
    field: FRST OPEN_F ;
    io: i;
    '}
    eState	:	E_ValvePositionState := INVALID;

    {attribute 'pytmc' := '
    pv: STATE;
    field: ZRST Vented;
    field: ONST At Vacuum;
    field: TWST Differential Pressure;
    field: THST Lost Vacuum;
    field: FRST Ext Fault;
    field: FVST AT Vacuum;
    field: SXST Triggered;
    field: SVST Vacuum Fault;
    field: EIST Close Timeout;
    field: NIST Open Timeout;
    io: i;
    '}
    eVGC_State : E_VGC;

(* Error *)

    {attribute 'pytmc' := '
    pv: ERROR;
    field: ZNAM NO ERROR ;
    field: ONAM ERROR PRESENT ;
    io: o;
    '}
    bErrorPresent : BOOL;
    iErrorCode: INT;
    {attribute 'pytmc' := '
    pv: ErrMsg;
    io: o;
    '}
    sErrorMessage: STRING;
    {attribute 'pytmc' := '
    pv: LOGGER;
    io: io;
    field: ZNAM OFF ;
    field: ONAM ON ;
    '}
    xLog : BOOL:=TRUE;

END_STRUCT
END_TYPE

// ---- DUTs/Valves/ST_VFS.TcDUT
TYPE ST_VFS EXTENDS ST_ValveBase:
STRUCT

(* Interlock *)
    {attribute 'pytmc' := '
    pv: TRIG;
    field: ZNAM TRIG_OFF;
    field: ONAM TRIG_ON;
    io: i ;
    '}
    i_xTrigger : BOOL;
(* Commands *)
    {attribute 'pytmc' := '
    pv: CLS_SW;
    field: ZNAM FALSE;
    field: ONAM CLOSE;
    io: io ;
    '}
    xCLS_SW AT%Q*:BOOL; (*external open signal e.g epics*)

(* Alarm Outputs *)
    {attribute 'pytmc' := '
    pv: ERR_Ext;
    field: ZNAM NO ERROR ;
    field: ONAM External error present ;
    io: i;
    '}
    xERR_ExtFault		: 	BOOL;
    {attribute 'pytmc' := '
    pv: VAC_FAULT_OK;
    field: ZNAM FAULT ;
    field: ONAM FAULT OK;
    io: i ;
    '}
    i_xVAC_FAULT_OK : BOOL; (*Valve Vacuum OK, is set to False when there is Vacuum Fault*)


(*ILK Devices*)
    {attribute 'pytmc' := '
    pv: GFS;
    io: i;
    '}
    sGFS: String;

    {attribute 'pytmc' := '
    pv: VETO_DEVICE;
    io: i;
    '}
    sVetoDeviceName: STRING;

END_STRUCT
END_TYPE

// ---- DUTs/Valves/ST_VGC_2S.TcDUT
TYPE ST_VGC_2S EXTENDS ST_VGC:
STRUCT
    {attribute 'pytmc' := '
    pv: AT_VAC_SP_DS;
    io: o;
    field: HOPR 1000
    field: LOPR 0
    field: PREC 2
    field: EGU "TORR"
    autosave_pass1: VAL DESC
    '}
    rAT_VAC_SP_DS	:	REAL := 0.000001;	// Interlock setpoint for gauges on the downstream side of the valve
    {attribute 'pytmc' := '
    pv: AT_VAC_HYS_DS;
    io: o;
    field: HOPR 1000
    field: LOPR 0
    field: PREC 2
    field: EGU "TORR"
    autosave_pass1: VAL DESC
    '}
    rAT_VAC_HYS_DS	:	REAL :=0.000001;	// Hysteresis of the vacuum sp downstream
    rAT_VAC_SP_LAST_DS :	REAL :=0.000001 ;
END_STRUCT
END_TYPE

// ---- DUTs/Valves/ST_VRC_NO.TcDUT
TYPE ST_VRC_NO EXTENDS ST_ValveBase:
STRUCT
(* Readbacks *)
    //In case VRC is normally open
    {attribute 'pytmc' := '
    pv: CLS_OK;
    field: ONAM TRUE;
    field: ZNAM FALSE;
    io: i;
    '}
    xCLS_OK : BOOL := TRUE;
    {attribute 'pytmc' := '
    pv: CLS_SW ;
    field: ONAM CLOSE;
    field: ZNAM OPEN;
    io: io ;
    '}
    pv_xCLS_SW	: BOOL;

    {attribute 'pytmc' := '
    pv: CLS_DO ;
    field: ONAM CLOSE;
    field: ZNAM OPEN;
    io: io ;
    '}
    q_xCLS_DO	: BOOL;
    {attribute 'pytmc' := '
    pv: FORCE_CLS;
    field: ONAM FORCE CLOSE;
    field: ZNAM FALSE;
    io: io;
    '}
    pv_xOvrdCls	:	BOOL;

END_STRUCT
END_TYPE

// ---- DUTs/Valves/ST_VWC_NO.TcDUT
TYPE ST_VWC_NO EXTENDS ST_VGC:
STRUCT
(* Readbacks *)
    //In case VRC is normally open
    {attribute 'pytmc' := '
    pv: CLS_OK;
    field: ONAM CLOSE;
    field: ZNAM OPEN;
    io: i;
    '}
    xCLS_OK : BOOL := TRUE;
    {attribute 'pytmc' := '
    pv: CLS_SW ;
    field: ONAM CLOSE;
    field: ZNAM OPEN;
    io: io ;
    '}
    pv_xCLS_SW	: BOOL;
    {attribute 'pytmc' := '
    pv: FORCE_CLS;
    field: ONAM FORCE CLOSE;
    field: ZNAM FALSE;
    io: io;
    '}
    pv_xOvrdCls	:	BOOL;

END_STRUCT
END_TYPE

// ---- DUTs/Valves/ST_VVC.TcDUT
TYPE ST_VVC :
STRUCT

(* Inputs *)

    {attribute 'pytmc' := '
    pv: OPN_SW;
    field: ZNAM CLOSE;
    field: ONAM OPEN;
    io: io;
    '}
    pv_xOPN_SW	: BOOL;
    {attribute 'pytmc' := '
    pv:FORCE_OPN;
    field: ZNAM FALSE;
    field: ONAM FORCE OPEN;
    io: io;
    '}
    xOvrdOpn	:	BOOL;
    {attribute 'pytmc' := '
    pv: OVRD_ON;
    field: ZNAM Override OFF ;
    field: ONAM Override ON;
    io: io;
    '}
    xOverrideMode	:	BOOL; (* Shows the override status of this valve *)
    {attribute 'pytmc' := '
    pv: OPN_OK;
    field: ZNAM OPN ILK NOT OK ;
    field: ONAM OPN ILK OK ;
    io: i;
    '}
    xOPN_OK	: BOOL;

(* Outputs *)
    {attribute 'pytmc' := '
    pv: OPN_DO;
    field: ZNAM CLOSE;
    field: ONAM OPEN;
    io: i;
    '}
    q_xOPN_DO	: BOOL;

END_STRUCT
END_TYPE

// ---- DUTs/Valves/ST_VCC_NO.TcDUT
TYPE ST_VCC_NO:
STRUCT

(* A normally open valve needs permission to close! *)
(* Inputs *)
    {attribute 'pytmc' := '
    pv: CLS_SW ;
    field: ONAM CLOSE;
    field: ZNAM OPEN;
    io: io ;
    '}
    pv_xCLS_SW	: BOOL;
    {attribute 'pytmc' := '
    pv: FORCE_CLS;
    field: ZNAM FALSE;
    field: ONAM FORCE CLOSE;
    io: io;
    '}
    pv_xOvrdCls	:	BOOL;
    {attribute 'pytmc' := '
    pv: CLS_OK;
    field: ZNAM FALSE;
    field: ONAM CLS_OK;
    io: i;
    '}
    xCLS_OK	: BOOL;

    {attribute 'pytmc' := '
    pv: OVRD_ON;
    field: ZNAM Override OFF ;
    field: ONAM Override ON;
    io: io
    '}
    xOverrideMode	:	BOOL; (* Shows the override status of this valve *)

(* Outputs *)
    {attribute 'pytmc' := '
    pv: CLS_DO;
        field: ZNAM FALSE;
    field: ONAM TRUE;
    io: i;
    '}
    xCLS_DO	: BOOL;

END_STRUCT
END_TYPE

// ---- DUTs/Valves/ST_VCN.TcDUT
TYPE ST_VCN :
STRUCT
    (* VCN - Valve Controlled Needle
    Used for Pfeiffer EVR 116 needle valves *)
    {attribute 'pytmc' := '
    pv: OPN_SW;
    field: ZNAM CLOSE;
    field: ONAM OPEN;
    io: io ;
    '}
    xOPN_SW	: BOOL;
    {attribute 'pytmc' := '
    pv: POS_RDBK;
    io: i;
    '}
    // Inputs
    i_iPosition	:	REAL; //Position readback (if it exists)

    // Outputs
    {attribute 'pytmc' := '
    pv: POS_AO_R;
    io: i ;
    '}
    q_iRawPosition	:	INT; //Position control
    //For the EVR 116 this is 0-10V analog 0.4 closed to 9.1 Closed

    //Softvariables
    {attribute 'pytmc' := '
    pv: ILK_OK;
    field: ZNAM NOT OK ;
    field: ONAM OK ;
    io: i;
    '}
    xIlkOK	:	BOOL := FALSE; // Interlock Bit

    {attribute 'pytmc' := '
    pv: ILK_SP;
    io: o;
    field: HOPR 1000
    field: LOPR 0
    field: PREC 2
    field: EGU "TORR"
    autosave_pass1: VAL DESC
    '}
    rIlk_SP	:	REAL := 0.0005;	// Interlock setpoint for gauges on both sides of valve

    {attribute 'pytmc' := '
    pv: Limit;
    io: io;
    autosave_pass1: VAL DESC
    '}
    rUpperLimit	:	REAL:=100; // Percentage//Upper limit on valve open
    {attribute 'pytmc' := '
    pv: POS_REQ;
    io: io;
    '}
    rReqPosition	:	REAL; //Requested position (0.0-100.0%)
    {attribute 'pytmc' :=  '
    pv: STATE ;
    field: ZRST Close ;
    field: ONST Open;
    field: TWST PressureControl ;
    field: THST ManualControl ;
    io: io
    '}
    eValveControl	:	E_VCN := CloseValve; // Valve control state

    ftIlk	:	F_TRIG;

END_STRUCT
END_TYPE

// ---- DUTs/Valves/ST_VGC.TcDUT
TYPE ST_VGC EXTENDS ST_ValveBase:
STRUCT


(* Interlocks *)

    {attribute 'pytmc' := '
    pv: DP_OK;
    field: ZNAM DP NOT OK ;
    field: ONAM DP OK ;
    io: i;
    '}
    xDP_OK	:	BOOL;	(* Managed by the VGC function (FB_VGC) *)// Indicates the valve can be opened because the differential pressure is low enough

    {attribute 'pytmc' := '
    pv: AT_VAC_SP;
    io: o;
    field: HOPR 1000
    field: LOPR 0
    field: PREC 2
    field: EGU "TORR"
    autosave_pass1: VAL DESC
    '}
    rAT_VAC_SP	:	REAL := 0.000001;	// Interlock setpoint for gauges on both sides of valve
    rAT_VAC_SP_LAST	:	REAL :=0.000001 ;	// Interlock setpoint for gauges on both sides of valve
    {attribute 'pytmc' := '
    pv: AT_VAC_HYS;
    io: o;
    field: HOPR 1000
    field: LOPR 0
    field: PREC 2
    field: EGU "TORR"
    autosave_pass1: VAL DESC
    '}
    rAT_VAC_HYS	:	REAL :=0.0000012;	// Hysteresis of the vacuum sp, default 20% above the SP
    {attribute 'pytmc' := '
    pv: HYST_PERC ;
    io: o;
    autosave_pass1: VAL DESC
    '}
    rHYST_PERC	:	REAL := 0.80;	// Hysteresis percentage

    {attribute 'pytmc' := '
    pv: AT_VAC ;
    field: ZNAM NOT AT VAC ;
    field: ONAM AT VAC ;
    io: i;
    '}
    xAT_VAC	:	BOOL;	//At vacuum setpoint


(* Alarm Outputs *)
    {attribute 'pytmc' := '
    pv: ERR_DifPres;
    field: ZNAM NO ERROR ;
    field: ONAM Diffrential error present ;
    io: i;
    '}
    xERR_DifPres		: 	BOOL;
    {attribute 'pytmc' := '
    pv: ERR_SP;
    field: ZNAM NO ERROR ;
    field: ONAM Setpoint error present ;
    io: i;
    '}
    xERR_SP			: 	BOOL;
    {attribute 'pytmc' := '
    pv: ERR_Ext;
    field: ZNAM NO ERROR ;
    field: ONAM External error present ;
    io: i;
    '}
    xERR_ExtFault		: 	BOOL;
    xAlmSum			: 	BOOL;
    sDevName :STRING;
(*ILK Devices*)
{attribute 'pytmc' := '
    pv: ILK_DEVICE_US;
    io: i;
    '}
    sIlkUSDeviceName: STRING;
    {attribute 'pytmc' := '
    pv: ILK_DEVICE_DS;
    io: i;
    '}
    sIlkDSDeviceName: STRING;

END_STRUCT
END_TYPE

// ---- DUTs/Valves/ST_VRC.TcDUT
TYPE ST_VRC EXTENDS ST_ValveBase:
STRUCT
(* Readbacks *)
    //In case VRC is normally open
    {attribute 'pytmc' := '
    pv: CLS_OK;
    io: i;
    '}
    xCLS_OK : BOOL := TRUE;

END_STRUCT
END_TYPE

// ---- DUTs/Valves/VAT590/EtherCAT Interface/E_ControlMode.TcDUT
{attribute 'qualified_only'}
{attribute 'strict'}
TYPE E_ControlMode :
(
    Init := 0,
    Synch := 1,
    ManualControl := 2,
    CloseValve := 3,
    OpenValve := 4,
    PressureControl := 5,
    HoldValve := 6,
    LearnProcedure := 7,
    InterlockOpen := 8,
    InterlockClose := 9,
    MaintenanceOpen := 10,
    MaintenanceClose := 11,
    PowerFailure := 12,
    Safety := 13,
    FatalError := 14
) USINT := Init;
END_TYPE

// ---- DUTs/Valves/VAT590/EtherCAT Interface/E_ControlModeSP.TcDUT
{attribute 'qualified_only'}
{attribute 'strict'}
TYPE E_ControlModeSP :
(
    ManualControl := 2,
    CloseValve := 3,
    OpenValve := 4,
    PressureControl := 5,
    HoldValve := 6,
    LearnProcedure := 7
) USINT := CloseValve;
END_TYPE

// ---- DUTs/Valves/VAT590/EtherCAT Interface/E_FatalErrors.TcDUT
{attribute 'qualified_only'}
{attribute 'strict'}
TYPE E_FatalErrors :
(
    NO_FATAL_ERROR := 0,
    NoStopDetectedSynch := 20,
    ValveBlockedSynch := 21,
    ValveBlocked := 22,
    StepLossSynch := 25,
    MotorDriverFault := 40
) UINT := NO_FATAL_ERROR;
END_TYPE

// ---- DUTs/Valves/VAT590/EtherCAT Interface/ST_ExtendedWarnings.TcDUT
TYPE ST_ExtendedWarnings :
STRUCT
    Bit0RemoteControlNotPossible: BIT;
    Bit1ControlModeSPNotAllowed : BIT;
    Bit2ZeroDisabled : BIT;
    Bit3PFODeactivated : BIT;
    Bit4Reserved : BIT;
    Bit5PressureSPOutOfRange : BIT;
    Bit6PositionSPOutOfRange : BIT;
    Bit7Reserved : BIT;
    Bit8Reserved : BIT;
    Bit9Reserved : BIT;
    Bit10CtrlSPOutOfRange : BIT;
    Bit11GeneralCtrlSPOutOfRange : BIT;
    Bit12ProcDataSettingsNotvalid : BIT;
    Bit13Reserved5 : BIT;
    Bit14Reserved6 : BIT;
    Bit15Reserved7 : BIT;
END_STRUCT
END_TYPE

// ---- DUTs/Valves/VAT590/EtherCAT Interface/ST_GeneralControlSP.TcDUT
TYPE ST_GeneralControlSP :
STRUCT
    Bit0ExecuteZero: BIT;
    Bit1Reserved : BIT;
    Bit2PingPongTxBit : BIT;
    Bit3Reserved : BIT;
    Bit4AccessMode : BIT;
    Bit5Reserved : BIT;
    Bit6Reserved : BIT;
    Bit7Reserved : BIT;
    Bit8Reserved : BIT;
    Bit9Reserved : BIT;
    Bit10Reserved : BIT;
    Bit11Reserved : BIT;
    Bit12Reserved : BIT;
    Bit13Reserved : BIT;
    Bit14Reserved : BIT;
    Bit15Reserved : BIT;
END_STRUCT
END_TYPE

// ---- DUTs/Valves/VAT590/EtherCAT Interface/ST_GeneralStatus.TcDUT
TYPE ST_GeneralStatus :
STRUCT
    Bit0FieldBusDatavalid: BIT;
    Bit1ZeroExecuted : BIT;
    Bit2PingPongRxBit : BIT;
    Bit3PressureSimulation : BIT;
    Bit4PressureSPReached : BIT;
    Bit5Reserved : BIT;
    Bit6Reserved : BIT;
    Bit7AccessModeBit0 : BIT;
    Bit8AccessModeBit1 : BIT;
    Bit9WarningsActive : BIT;
    Bit10Reserved : BIT;
    Bit11Reserved : BIT;
    Bit12Reserved : BIT;
    Bit13Reserved : BIT;
    Bit14Reserved : BIT;
    Bit15Reserved : BIT;
END_STRUCT
END_TYPE

// ---- DUTs/Valves/VAT590/EtherCAT Interface/ST_GeneralWarnings.TcDUT
TYPE ST_GeneralWarnings :
STRUCT
    Bit0ServiceRequest: BIT;
    Bit1Reserved : BIT;
    Bit2Reserved : BIT;
    Bit3PowerFailureBattery : BIT;
    Bit4Reserved : BIT;
    Bit5Reserved : BIT;
    Bit6Reserved : BIT;
    Bit7Reserved : BIT;
    Bit8Reserved : BIT;
    Bit9Reserved : BIT;
    Bit10SensMeasUnitFault : BIT;
    Bit11Reserved : BIT;
    Bit12Reserved : BIT;
    Bit13Reserved : BIT;
    Bit14Reserved : BIT;
    Bit15Reserved : BIT;
END_STRUCT
END_TYPE

// ---- DUTs/Valves/VAT590/E_VAT590_AccessMode.TcDUT
{attribute 'qualified_only'}
{attribute 'strict'}
TYPE E_VAT590_AccessMode :
(
    LOCAL := 0,
    REMOTE := 1,
    LOCKED := 2
) USINT := REMOTE;
END_TYPE

// ---- DUTs/Valves/VAT590/E_VAT590_PID_CTRL.TcDUT
{attribute 'qualified_only'}
{attribute 'strict'}
TYPE E_VAT590_PID_CTRL :
(
    ADAPTIVE_DS := 0,
    FIXED_1 := 1,
    FIXED_2 := 2,
    SOFT_PUMP := 3
) USINT := FIXED_1;
END_TYPE

// ---- DUTs/Valves/VAT590/E_VCN_VAT590.TcDUT
{attribute 'qualified_only'}
{attribute 'strict'}
TYPE E_VCN_VAT590 :
(
    ManualControl := 0,
    CloseValve := 1,
    OpenValve := 2,
    PressureControl := 3,
    HoldValve := 4
) USINT := CloseValve;
END_TYPE

// ---- DUTs/Valves/VAT590/ST_CoEIndSub.TcDUT
TYPE ST_CoEIndSub :
STRUCT
    nIndex : WORD;
    nSubIndex : BYTE;
END_STRUCT
END_TYPE

// ---- DUTs/Valves/VAT590/ST_VAT590_COE.TcDUT
TYPE ST_VAT590_COE :
STRUCT
    {attribute 'pytmc' := '
    pv: PID_CTRL
    io: io
    '}
    ePIDCtrl: E_VAT590_PID_CTRL;
    (*Adaptive Downstream Parameters*)
    {attribute 'pytmc' := '
    pv: SENS_DELAY_AD
    io: io
    field: EGU "s"
    field: DRVL 0.0
    field: DRVH 1.0
    '}
    fSensorDelay_AD : REAL;
    {attribute 'pytmc' := '
    pv: RAMP_TIME_AD
    io: io
    field: EGU "s"
    field: DRVL 0.0
    field: DRVH 1000000.0
    '}
    fRampTime_AD : REAL;
    {attribute 'pytmc' := '
    pv: RAMP_MODE_AD
    io: io
    field: ZNAM CONST_TIME
    field: ONAM CONST_SLOPE
    '}
    bRampMode_AD : BOOL;
    {attribute 'pytmc' := '
    pv: GAIN_FACTOR_AD
    io: io
    field: PREC 4
    field: DRVL 0.0001
    field: DRVH 7.5
    '}
    fGainFactor_AD : REAL;
    (*Fixed 1 Parameters*)
    {attribute 'pytmc' := '
    pv: RAMP_TIME_FIX1
    io: io
    field: EGU "s"
    field: DRVL 0.0
    field: DRVH 1000000.0
    '}
    fRampTime_FIX1 : REAL;
    {attribute 'pytmc' := '
    pv: RAMP_MODE_FIX1
    io: io
    field: ZNAM CONST_TIME
    field: ONAM CONST_SLOPE
    '}
    bRampMode_FIX1 : BOOL;
    {attribute 'pytmc' := '
    pv: CTRL_DIR_FIX1
    io: io
    field: ZNAM DOWNSTREAM
    field: ONAM UPSTREAM
    '}
    bCtrlDir_FIX1 : BOOL;
    {attribute 'pytmc' := '
    pv: PGAIN_FIX1
    io: io
    field: DRVL 0.001
    field: DRVH 100.0
    '}
    fPGain_FIX1 : REAL;
    {attribute 'pytmc' := '
    pv: IGAIN_FIX1
    io: io
    field: DRVL 0.0
    field: DRVH 100.0
    '}
    fIGain_FIX1 : REAL;
    (*Fixed 2 Parameters*)
    {attribute 'pytmc' := '
    pv: RAMP_TIME_FIX2
    io: io
    field: EGU "s"
    field: DRVL 0.0
    field: DRVH 1000000.0
    '}
    fRampTime_FIX2 : REAL;
    {attribute 'pytmc' := '
    pv: RAMP_MODE_FIX2
    io: io
    field: ZNAM CONST_TIME
    field: ONAM CONST_SLOPE
    '}
    bRampMode_FIX2 : BOOL;
    {attribute 'pytmc' := '
    pv: CTRL_DIR_FIX2
    io: io
    field: ZNAM DOWNSTREAM
    field: ONAM UPSTREAM
    '}
    bCtrlDir_FIX2 : BOOL;
    {attribute 'pytmc' := '
    pv: PGAIN_FIX2
    io: io
    field: DRVL 0.001
    field: DRVH 100.0
    '}
    fPGain_FIX2 : REAL;
    {attribute 'pytmc' := '
    pv: IGAIN_FIX2
    io: io
    field: DRVL 0.0
    field: DRVH 100.0
    '}
    fIGain_FIX2 : REAL;
    (*Soft Pump Parameters*)
    {attribute 'pytmc' := '
    pv: RAMP_TIME_SP
    io: io
    field: EGU "s"
    field: DRVL 0.0
    field: DRVH 1000000.0
    '}
    fRampTime_SP : REAL;
    {attribute 'pytmc' := '
    pv: RAMP_MODE_SP
    io: io
    field: ZNAM CONST_TIME
    field: ONAM CONST_SLOPE
    '}
    bRampMode_SP : BOOL;
    {attribute 'pytmc' := '
    pv: PGAIN_SP
    io: io
    field: DRVL 0.001
    field: DRVH 100.0
    '}
    fPGain_SP : REAL;
    (*Position Limit Parameters*)
    {attribute 'pytmc' := '
    pv: POSITION_LIMIT_OPN
    io: io
    field: EGU "%"
    field: DRVL 0.0
    field: DRVH 100.0
    '}
    fPositionLimitOpen : REAL;
    {attribute 'pytmc' := '
    pv: POSITION_LIMIT_OPN_CTRL
    io: io
    field: EGU "%"
    field: DRVL 0.0
    field: DRVH 100.0
    '}
    fPositionLimitOpenControl : REAL;
END_STRUCT
END_TYPE

// ---- DUTs/Valves/VAT590/ST_VAT590_STATUS.TcDUT
TYPE ST_VAT590_STATUS :
STRUCT
    {attribute 'pytmc' :=  '
        pv: CTRL_MODE
        io: i
    '}
    eControlMode : E_ControlMode; // Valve control mode readback
    {attribute 'pytmc' :=  '
        pv: FATAL_ERR
        io: i
    '}
    eFatalErrors : E_FatalErrors; // Valve Fatal Error status readback
    (*General Status readback*)
    {attribute 'pytmc' := '
        pv: GEN_STATUS:ECAT_DATA_VALID
        io: i
        field: ZNAM NOT_VALID
        field: ONAM VALID
        field: ZSV MAJOR
        field: OSV NO_ALARM
    '}
    bFieldBusDatavalid: BOOL;
    {attribute 'pytmc' := '
        pv: GEN_STATUS:ZERO_EXECUTED
        io: i
        field: ZNAM NOT_EXECUTED
        field: ONAM EXECUTED
        field: ZSV NO_ALARM
        field: OSV NO_ALARM
    '}
    bZeroExecuted : BOOL;
    {attribute 'pytmc' := '
        pv: GEN_STATUS:ECAT_RxBIT
        io: i
        field: ZNAM NOT_INVERTED
        field: ONAM INVERTED
        field: ZSV NO_ALARM
        field: OSV NO_ALARM
    '}
    bPingPongRxBit : BOOL;
    {attribute 'pytmc' := '
        pv: GEN_STATUS:PRES_SIM
        io: i
        field: ZNAM OFF
        field: ONAM ON
        field: ZSV NO_ALARM
        field: OSV NO_ALARM
    '}
    bPressureSimulation : BOOL;
    {attribute 'pytmc' := '
        pv: GEN_STATUS:PRES_SP_REACHED
        io: i
        field: ZNAM NOT_AT_SP
        field: ONAM AT_SP
        field: ZSV NO_ALARM
        field: OSV NO_ALARM
    '}
    bPressureSPReached : BOOL;
    {attribute 'pytmc' := '
        pv: GEN_STATUS:WARN_STATUS
        io: i
        field: ZNAM NOT_ACTIVE
        field: ONAM ACTIVE
        field: ZSV NO_ALARM
        field: OSV MAJOR
    '}
    bWarningsActive : BOOL;
    {attribute 'pytmc' :=  '
        pv: GEN_STATUS:REM_CTRL
        io: i
    '}
    eRemoteStatus : E_VAT590_AccessMode;
    (*General Warnings readback*)
    {attribute 'pytmc' := '
        pv: GEN_WARN:SERVICE_REQ
        io: i
        field: ZNAM OK
        field: ONAM SERVICE
        field: ZSV NO_ALARM
        field: OSV MAJOR
    '}
    bServiceRequest: BOOL;
    {attribute 'pytmc' := '
        pv: GEN_WARN:POWER_FAIL_BATT
        io: i
        field: ZNAM READY
        field: ONAM NOT_READY
        field: ZSV NO_ALARM
        field: OSV MINOR
    '}
    bPowerFailureBattery : BOOL;
    {attribute 'pytmc' := '
        pv: GEN_WARN:ADC_UNIT_STATUS
        io: i
        field: ZNAM OK
        field: ONAM FAULT
        field: ZSV NO_ALARM
        field: OSV MAJOR
    '}
    bSensMeasUnitFault : BOOL;
    (*Extended Warnings readback*)
    {attribute 'pytmc' := '
        pv: EXT_WARN:REM_NOT_POSSIBLE
        io: i
        field: ZNAM ENABLED
        field: ONAM DISABLED
        field: ZSV NO_ALARM
        field: OSV MINOR
    '}
    bRemoteControlNotPossible: BOOL;
    {attribute 'pytmc' := '
        pv: EXT_WARN:CTRL_SP_NOT_ALLOWED
        io: i
        field: ZNAM ENABLED
        field: ONAM DISABLED
        field: ZSV NO_ALARM
        field: OSV MINOR
    '}
    bControlModeSPNotAllowed : BOOL;
    {attribute 'pytmc' := '
        pv: EXT_WARN:ZERO_STATUS
        io: i
        field: ZNAM ENABLED
        field: ONAM DISABLED
        field: ZSV NO_ALARM
        field: OSV MINOR
    '}
    bZeroDisabled : BOOL;
    {attribute 'pytmc' := '
        pv: EXT_WARN:PFO_STATUS
        io: i
        field: ZNAM ENABLED
        field: ONAM DISABLED
        field: ZSV NO_ALARM
        field: OSV MINOR
    '}
    bPFODeactivated : BOOL;
    {attribute 'pytmc' := '
        pv: EXT_WARN:PRES_SP_OOR
        io: i
        field: ZNAM OK
        field: ONAM FAULT
        field: ZSV NO_ALARM
        field: OSV MAJOR
    '}
    bPressureSPOutOfRange : BOOL;
    {attribute 'pytmc' := '
        pv: EXT_WARN:POS_SP_OOR
        io: i
        field: ZNAM OK
        field: ONAM FAULT
        field: ZSV NO_ALARM
        field: OSV MAJOR
    '}
    bPositionSPOutOfRange : BOOL;
    {attribute 'pytmc' := '
        pv: EXT_WARN:CTRL_SP_OOR
        io: i
        field: ZNAM OK
        field: ONAM FAULT
        field: ZSV NO_ALARM
        field: OSV MAJOR
    '}
    bCtrlSPOutOfRange : BOOL;
    {attribute 'pytmc' := '
        pv: EXT_WARN:GENCTRL_SP_OOR
        io: i
        field: ZNAM OK
        field: ONAM FAULT
        field: ZSV NO_ALARM
        field: OSV MAJOR
    '}
    bGeneralCtrlSPOutOfRange : BOOL;
    {attribute 'pytmc' := '
        pv: EXT_WARN:PROC_DATA_NOT_VALID
        io: i
        field: ZNAM OK
        field: ONAM FAULT
        field: ZSV NO_ALARM
        field: OSV MAJOR
    '}
    bProcDataSettingsNotvalid : BOOL;
END_STRUCT
END_TYPE

// ---- DUTs/Valves/VAT590/ST_VCN_VAT590.TcDUT
TYPE ST_VCN_VAT590 :
STRUCT
    (* VCN - Valve Controlled Needle
    Used for VAT590 needle valves *)
    {attribute 'pytmc' := '
    pv: POS_RAW
    io: i
    '}
    nRawPosition : DINT; //Position readback
    {attribute 'pytmc' := '
    pv: PRES_RAW
    io: i
    '}
    nRawPressure : DINT; //Pressure readback
    {attribute 'pytmc' := '
    pv: PRES_TORR
    field: EGU "TORR"
    io: i
    '}
    fPressure : REAL; //Pressure readback in Torr units
    {attribute 'pytmc' := '
    pv: POS_SP
    io: i
    '}
    nPositionSP : DINT; //Position setpoint readback
    {attribute 'pytmc' := '
    pv: PRES_SP
    io: i
    '}
    nPressureSP : DINT; //Pressure setpoint readback
    {attribute 'pytmc' := '
    pv: ILK_OK
    field: ZNAM NOT OK
    field: ONAM OK
    field: ZSV MAJOR
    field: OSV NO_ALARM
    io: i
    '}
    bIlkOK : BOOL := FALSE; //Interlock Bit status
    {attribute 'pytmc' := '
    pv: POS_LIMIT
    io: io
    autosave_pass1: VAL DESC
    '}
    fPosSetLimit	: REAL := 100; //Percentage Upper limit on valve open
    {attribute 'pytmc' := '
    pv: PRES_SET_LIMIT
    io: io
    autosave_pass1: VAL DESC
    '}
    fPresSetLimit	: REAL := 1E-2; //Upper limit for pressure control
    {attribute 'pytmc' := '
    pv: PRES_RDBK_LIMIT
    io: io
    autosave_pass1: VAL DESC
    '}
    fPresRdbkLimit : REAL := 1E-4;  //Upper limit for pressure reading before valve close
    {attribute 'pytmc' := '
    pv: POS_REQ
    field: DRVL 0.0
    field: DRVH 100.0
    io: io
    '}
    fReqPosition : REAL; //Requested position (0.0-100.0%)
    {attribute 'pytmc' := '
    pv: PRES_REQ
    field: EGU "TORR"
    io: io;
    '}
    fReqPressure : REAL; //Requested pressure in Torr units
    {attribute 'pytmc' :=  '
    pv: STATE
    io: io
    '}
    eValveControl : E_VCN_VAT590; //Valve control mode
    {attribute 'pytmc' := '
    pv:
    '}
    stValveStatus : ST_VAT590_STATUS; //All Valve status readbacks
    {attribute 'pytmc' :=  '
    pv: REM_CTRL
    io: io
    '}
    eRemoteControl : E_VAT590_AccessMode; //Select remote control mode
    {attribute 'pytmc' := '
    pv: ZERO
    io: io
    '}
    bZero : BOOL; //Activate Zero function bit
    {attribute 'pytmc' := '
    pv: COE_PARAM
    '}
    stCoeParameters : ST_VAT590_COE; //Coe Parameters
    {attribute 'pytmc' := '
    pv: COE_ERROR
    field: ZNAM OK
    field: ONAM ERROR
    field: ZSV NO_ALARM
    field: OSV MINOR
    io: i
    '}
    bCoeError : BOOL; //Coe Interface Error
    {attribute 'pytmc' := '
    pv: COE_RESET
    io: io
    '}
    bResetCoeError : BOOL; //Reset Coe Interface Error
    {attribute 'pytmc' := '
    pv: ETHCAT_COMM_STATUS
    field: ZNAM OK
    field: ONAM ERROR
    field: ZSV NO_ALARM
    field: OSV MAJOR
    io: i
    '}
    bValveEthCatStatus : BOOL; //Status of the Ethercat Communication with device
END_STRUCT
END_TYPE

// ---- GVLs/Constants.TcGVL
VAR_GLOBAL CONSTANT
    gc_iSizeOfGGOArray : INT := 50;
    gc_GaugeValidState :	INT := 4;
END_VAR

// ---- GVLs/Global_Variables.TcGVL
VAR_GLOBAL
    g_iSizeOfGGOArray : INT := 50;

    g_stSystem	:	ST_System(*System_Struct*):= (
        xFirstScan := TRUE
    );

    g_DummyVG	:	ST_VG;


     fbGetCurTaskIdx : GETCURTASKINDEX;
     TaskInfo:PlcTaskSystemInfo;


END_VAR

// ---- GVLs/GVL_MacroSensorsParameters.TcGVL
VAR_GLOBAL CONSTANT
    gcMaxLVC4000	:	INT := 20; //maximum number of LVC4000 units per port
END_VAR

// ---- GVLs/GVL_PfeifferParameters.TcGVL
VAR_GLOBAL CONSTANT
    gcMaxPfeifferPumps	:	INT := 20; //maximum size of the Pfeiffer turbo pump array for a single port
END_VAR

// ---- Version/Global_Version.TcGVL
{attribute 'TcGenerated'}
{attribute 'no-analysis'}
{attribute 'linkalways'}
// This function has been automatically generated from the project information.
VAR_GLOBAL CONSTANT
    {attribute 'const_non_replaced'}
    stLibVersion_LCLS_Vacuum : ST_LibVersion := (iMajor := 2, iMinor := 6, iBuild := 6, iRevision := 0, nFlags := 1, sVersion := '2.6.6');
END_VAR

// ---- POUs/Functions/Valves/Interfaces/ITF_Valve.TcIO
INTERFACE ITF_Valve

END_INTERFACE

// ---- UnitTests/PRG_Test.TcPOU
PROGRAM PRG_Test
VAR
    //fb_VGC_Test: FB_VGC_Test;
    //fb_VRC_Test: FB_VRC_Test;
    //fb_PIP_Test: FB_PIP_Test;
    //fb_PTM_Test: FB_PTM_Test;
    //fb_GPI_Test:FB_GPI_Test;
    fb_GHC_Test:FB_GHC_Test;

    TotalTests : INT:=0;
END_VAR


TcUnit.RUN();

END_PROGRAM

// ---- UnitTests/Gauges/FB_GHC_Test.TcPOU
FUNCTION_BLOCK FB_GHC_Test EXTENDS TcUnit.FB_TestSuite
VAR_INPUT
END_VAR
VAR_OUTPUT
END_VAR
VAR
    PG : ST_VG;
    fb_MKS355: FB_MKS355;
    i_iPRESS_R AT %Q* :INT;
    cycle:INT :=0;
END_VAR

M_INIT();
M_Interlock();
M_CheckRange();
//M_SelfProtection();
cycle:=cycle+1;


fb_MKS355(PG:=PG, IG=>);

METHOD M_CheckRange
VAR
    Expected:REAL;
    Actual:REAL;
    eStateExpected: E_PressureState;
    eStateActual: E_PressureState;
END_VAR
TEST('Check_Range');
Case This^.cycle of
    12:
    THIS^.fb_MKS355.i_iPRESS_R_test :=  V_TO_INT(1);
    THIS^.fb_MKS355.PG.rPRESS := 1E-4;
    THIS^.fb_MKS355.PG.xPRESS_OK := TRUE;
    THIS^.fb_MKS355.M_HVE(TRUE);

    15:
    TEST('MKS355_Range_Valid');
    Expected :=1E-9 ;
    eStateExpected := Valid;
    Actual := THIS^.fb_MKS355.IG.rPRESS;
    eStateActual := THIS^.fb_MKS355.IG.eState;
    AssertTrue(THIS^.fb_MKS355.IG.xPRESS_OK, 'MKS355 xPRESS_OK is set to False');
    AssertEquals(eStateExpected,eStateActual,'MKS355 eState Fail');
    AssertEquals_REAL(Expected, Actual,1E-10, 'MKS355 rPress Fail');
    TEST_FINISHED_NAMED('MKS355_Range_Valid');

    20:
    THIS^.fb_MKS355.i_iPRESS_R_test :=  V_TO_INT(0.001);

    21:
    TEST('MKS355_Range_ValidLo');
    Expected :=1E-10;
    Actual := THIS^.fb_MKS355.IG.rPRESS;
    eStateExpected := ValidLo;
    eStateActual := THIS^.fb_MKS355.IG.eState;
    AssertTrue(THIS^.fb_MKS355.IG.xPRESS_OK, 'MKS355 xPRESS_OK is set to False');
    AssertEquals(eStateExpected,eStateActual,'MKS355 eState Fail');
    AssertEquals_REAL(Expected, Actual,1E-10, 'MKS355 rPress Fail');
    TEST_FINISHED_NAMED('MKS355_Range_ValidLo');


    24:
    THIS^.fb_MKS355.i_iPRESS_R_test :=  V_TO_INT(10);

    25:
    TEST('MKS355_Range_Off');
    Expected :=0 ;
    eStateExpected := Off;
    Actual := THIS^.fb_MKS355.IG.rPRESS;
    eStateActual := THIS^.fb_MKS355.IG.eState;
    AssertFalse(THIS^.fb_MKS355.IG.xPRESS_OK, 'MKS355 xPRESS_OK is set to True');
    AssertEquals(eStateExpected,eStateActual,'MKS355 eState Fail');
    AssertEquals_REAL(Expected, Actual,1, 'MKS355 rPress Fail');
    TEST_FINISHED_NAMED('MKS355_Range_Off');


END_CASE
END_METHOD

METHOD M_INIT
VAR
END_VAR
TEST('MKS355_Startup');
IF (cycle = 1) THEN
    THIS^.PG.rPRESS := 1E-4;
    THIS^.PG.xPRESS_OK := TRUE;
    THIS^.fb_MKS355(PG:=THIS^.PG, IG=>);
    THIS^.fb_MKS355.M_HVE(TRUE);
    AssertTrue(THIS^.fb_MKS355.IG.xHV_SW, 'MKS355 xHV_SW set to False');
ELSIF (cycle = 2) THEN
    THIS^.fb_MKS355(PG:=THIS^.PG, IG=>);
    AssertTrue(THIS^.fb_MKS355.IG.q_xHV_DIS, 'MKS355 q_xHV_DIS set to False');
    TEST_FINISHED_NAMED('MKS355_Startup');
End_IF;
END_METHOD

METHOD M_Interlock
VAR_INPUT
END_VAR
TEST('MKS355_Interlock_Active');
TEST('MKS355_Interlock_OK');
TEST('MKS355_Interlock_Lost');

CASE cycle OF

    3:
    THIS^.fb_MKS355.PG.rPRESS := 1E-1;
    THIS^.fb_MKS355.PG.xPRESS_OK := FALSE;
    fb_MKS355.M_HVE(FALSE);

    4:
    AssertFalse(THIS^.fb_MKS355.IG.xHV_SW, 'MKS355 xHV_SW set to True');
    AssertFalse(THIS^.fb_MKS355.IG.q_xHV_DIS, 'MKS355 q_xHV_DIS set to True');
    TEST_FINISHED_NAMED('MKS355_Interlock_Lost');

    5:
    THIS^.fb_MKS355.PG.rPRESS := 1E-4;
    THIS^.fb_MKS355.PG.xPRESS_OK := TRUE;
    fb_MKS355.M_HVE(TRUE);

    6:
    AssertTrue(THIS^.fb_MKS355.IG.xHV_SW, 'MKS355 xHV_SW set to False');
    AssertTrue(THIS^.fb_MKS355.IG.q_xHV_DIS, 'MKS355 q_xHV_DIS set to False');
    TEST_FINISHED_NAMED('MKS355_Interlock_OK');

END_CASE
END_METHOD

METHOD M_SelfProtection
VAR_INPUT
END_VAR
// Switching the Cold cathode backon
TEST('MKS355_Interlock_OK_1');
This^.PG.rPRESS := 1E-4;
This^.PG.xPRESS_OK := True;
fb_MKS355.M_HVE(TRUE);
THIS^.fb_MKS355(PG:=THIS^.PG, IG=>);
AssertTrue(THIS^.fb_MKS355.IG.xHV_SW, 'MKS355 xHV_SW set to False');
AssertFalse(THIS^.fb_MKS355.IG.q_xHV_DIS, 'MKS355 q_xHV_DIS set to True');
TEST_FINISHED_NAMED('MKS355_Interlock_OK_1');

TEST('MKS355_Self_Protection');
This^.PG.rPRESS := 1E-3;
This^.PG.xPRESS_OK := TRUE;
THIS^.fb_MKS355(PG:=THIS^.PG, IG=>);
AssertFalse(THIS^.fb_MKS355.IG.xHV_SW, 'MKS355 xHV_SW set to True');
AssertTrue(THIS^.fb_MKS355.IG.q_xHV_DIS, 'MKS355 q_xHV_DIS set to False');
TEST_FINISHED_NAMED('MKS355_Self_Protection');
END_METHOD

END_FUNCTION_BLOCK

// ---- POUs/Functions/Gauges/FB_MKS355.TcPOU
(* This function is for the Hot Cathode MKS 355.

This function provides ILK and Set Point Protection for the hot Cathode.
*)

FUNCTION_BLOCK FB_MKS355 EXTENDS FB_GaugeBase
VAR_IN_OUT

END_VAR
VAR_INPUT
    PG	:	ST_VG;
    tRecoverDelay:TIME:=T#600S; (*Delay Time after the first cycle to start the device. Default is 600S*)
END_VAR
VAR_OUTPUT
{attribute 'pytmc' := '
    pv:
    '}
    IG : ST_VG;
END_VAR
VAR
    rV : REAL;
    GaugeTurnOnTmr : TON;
    tStartupTimer:TON;
    iTermBits: UINT := 30518 ; // The terminal's maximum value in bits
    (*IOs to be linked*)
    /// Controls and I/Os
    i_iPRESS_R AT %I* :INT; // input Pressure // Link to analog Input
    q_xHV_DIS AT %Q* : BOOL; // Enable High Voltage when True // 'TcLinkTo' (EP2624) ^Output
    // only for EL and ES terminal
    i_xHV_ON AT %I*	: BOOL; //  True when High Voltage is on  // 'TcLinkTo' (EL1084) ^Input

    binit:BOOL:=TRUE;
END_VAR

VAR CONSTANT
    vBase : REAL := 1.0;
    vDisconnected : REAL:= 0.001; //shift from 0 to eliminate single noise effect
    vTorr : REAL := 10;
    vGaugeOff: REAL := 10;
    rMinPressure: REAL := 1E-10;
    cDefaultPressure : REAL := 0;
    rDeadband : REAL :=1.0;
END_VAR

VAR PERSISTENT
    bWasOn : BOOL;
    bAutoRecover:BOOL;
    bAutoRecoverWrite:BOOL;
END_VAR

(*Startup time*)
IF (bInit) THEN
    tStartupTimer.IN:=TRUE;
    bInit :=FALSE;
END_IF
tStartupTimer(PT:=T#3S);

(* 355 Logarithmic Output Conversion, factory default configuration
   EL3174, EL3174-xxxx iTermbits 30518, 10V
*)
If (iTermBits=0) THEN iTermBits := 30518;END_IF
rV := 10*INT_TO_REAL(IG.i_iPRESS_R)/iTermBits;

(* Set Guage State based on the Analog voltage*)

IF rV <= vDisconnected AND IG.i_xHV_ON and IG.q_xHV_DIS THEN
    IG.eState := ValidLo;
    IG.rPRESS := rMinPressure;
ELSIF rV <= vDisconnected AND NOT IG.i_xHV_ON AND IG.q_xHV_DIS THEN
    IG.eState := GaugeDisconnected;
    IG.rPRESS := cDefaultPressure;
ELSIF rV > vDisconnected AND rV < (vGaugeOff -rDeadband) AND IG.i_xHV_ON AND IG.q_xHV_DIS THEN
    IG.eState := Valid;
    IG.rPRESS := LREAL_TO_REAL(EXPT(10,((rV*vBase)- vTorr)));
ELSIF rV >= (vGaugeOff -rDeadband) THEN
    IG.eState := Off;
    IG.rPRESS := cDefaultPressure;
ELSE
    IG.eState := OoR;
    IG.rPRESS := cDefaultPressure;
END_IF



(* Ion Gauge Protection Functions *)
(* If the PG pressure is greater than the VG.PRO_SP then the gauge is disabled *)
(* If the PG pressure is less than the VG.PRO_SP then the gauge is enabled *)
(* This FB also implements some hysteresis so the gauge doesn't have rapid power cycling while near the turn on boundary *)


IF PG.rPRESS <= IG.rPRO_SP AND PG.xPRESS_OK THEN
    IG.q_xHV_DIS := IG.xHV_SW;
    IG.xILKOk := TRUE;
ELSIF IG.q_xHV_DIS THEN
    IF IG.rPRESS > (IG.rPRO_SP + IG.rHYS_PR)  OR PG.rPRESS > (IG.rPRO_SP + IG.rHYS_PR) THEN
        IG.q_xHV_DIS := FALSE;
        IG.xHV_SW := FALSE;
    END_IF
ELSE
    IG.q_xHV_DIS := FALSE;
    IG.xHV_SW := FALSE;
    IG.xILKOk := FALSE;
END_IF

(* Pressure gauge OK checks *)

GaugeTurnOnTmr(IN:=IG.q_xHV_DIS, PT:=T#10S, Q=>IG.xTurnOnTime);

//Backwards compatibility
IG.xPRESS_OK := (IG.eState = Valid) OR (IG.eState = ValidLo) OR IG.xBAKEOUT;

(* Setpoint evaluation *)
IG.xAT_VAC := (IG.xPRESS_OK AND (IG.rPRESS < IG.rVAC_SP)) OR IG.xBAKEOUT AND (IG.eState = Valid) ;

ACT_Logger();
(*Soft IO Linking*)
// check ethercat Diagnostics
IO();
(*Load or save the persistent variables*)
ACT_Persistent();
(*Run Auto Recovery*)
ACT_Recover();

ACTION ACT_Logger:
// ILK logger
IF (IG.xLog) THEN
    IF NOT IG.xILKOk AND IG.q_xHV_DIS THEN
            fbLogger(sMsg:='Lost external interlock while gauge was on.', eSevr:=TcEventSeverity.Critical);
    END_IF


    // Log Action
    tAction(CLK:=   IG.xHV_SW);
    IF tAction.Q THEN fbLogger(sMsg:='Ion gauge commanded to switch on', eSevr:=TcEventSeverity.Info); END_IF



    //STATE Logger
    tState(CLK:=  ePrevState <> IG.eState);
    IF ePrevState <> IG.eState THEN
          CASE IG.eState OF
            ValidHi:
                fbLogger(sMsg:='Gauge pressure valid high.', eSevr:=TcEventSeverity.Info);
            ValidLo:
                fbLogger(sMsg:='Gauge pressure valid low.', eSevr:=TcEventSeverity.Info);
            Valid:
                fbLogger(sMsg:='Gauge pressure valid.', eSevr:=TcEventSeverity.Info);
            GaugeDisconnected:
                fbLogger(sMsg:='Gauge Disconnected.', eSevr:=TcEventSeverity.Critical);
            PressInvalid:
                fbLogger(sMsg:='Gauge pressure invalid.', eSevr:=TcEventSeverity.Warning);
            OoR:
                fbLogger(sMsg:='Gauge pressure out of range.', eSevr:=TcEventSeverity.Warning);
            Starting:
                fbLogger(sMsg:='Gauge starting.', eSevr:=TcEventSeverity.Info);
          END_CASE
          ePrevState := IG.eState;
          stateTimer.IN := TRUE;
      END_IF
END_IF
END_ACTION

ACTION ACT_Persistent:
(*On first PLC pass, load the persistent value into the structrue variable*)
IF (SUPER^.bRestorePersistentData) THEN
    SUPER^.bRestorePersistentData	:= FALSE;
    IF ( rVAC_SP <> 0) THEN
        IG.rVAC_SP := rVAC_SP;
    END_IF;
    IF ( rPRO_SP <> 0) THEN
        IG.rPRO_SP := rPRO_SP;
    END_IF;
    IF ( rHYS_PR <> 0) THEN
        IG.rHYS_PR := rHYS_PR;
    END_IF;
    IF ( bAutoRecoverWrite) THEN
        IG.xAutoOn := bAutoRecover;
    END_IF;
END_IF
(*Check if a new value has been written in the structure variable copy it to the persistent variable*)
IF NOT (IG.rVAC_SP = rVAC_SP)  THEN
    rVAC_SP := IG.rVAC_SP;
END_IF;

IF NOT (IG.rPRO_SP = rPRO_SP) THEN
    rPRO_SP:= IG.rPRO_SP;
END_IF;

IF NOT (IG.rHYS_PR = rHYS_PR) THEN
    rHYS_PR:= IG.rHYS_PR;
END_IF;

IF NOT(bAutoRecoverWrite) OR NOT (bAutoRecover = IG.xAutoOn) THEN
    bAutoRecover := IG.xAutoOn;
    bAutoRecoverWrite := TRUE;
END_IF;
stateTimer(PT:=T#10S);
IF (stateTimer.Q) THEN
    bWasOn := (IG.eState >=Valid );
    stateTimer.IN := FALSE;
    fbWritePersistentData(NETID:='', PORT:=851, START:=TRUE, TMOUT:=T#1s );
END_IF;
END_ACTION

ACTION ACT_Recover:
fbGetCurTaskIdx();
IF (TwinCAT_SystemInfoVarList._TaskInfo[fbGetCurTaskIdx.index].FirstCycle) THEN
    tRecover.IN := TRUE;
END_IF
tRecover(IN:= , PT:=tRecoverDelay);
IF NOT(bAutoRecoverWrite) OR (tRecover.Q AND bAutoRecover ) THEN
    This^.M_Recover();
    tRecover.IN := FALSE;
END_IF
END_ACTION

ACTION IO:
(*soft link inputs*)
IG.i_iPRESS_R:=	i_iPRESS_R;
IG.i_xHV_ON:= i_xHV_ON;
//IG.i_xDisc_Active:=i_xDisc_Active;
(*soft link outputs*)
q_xHV_DIS := IG.q_xHV_DIS;

IG.sPath := sPath;
IG.iAutoOnTimer:= TIME_TO_INT(tRecover.PT);
END_ACTION

METHOD M_HVE : BOOL
VAR_INPUT
        enable:bool; // set to true to enable, false to disable;
END_VAR
this^.IG.xHV_SW:= enable;
END_METHOD

METHOD M_Recover : BOOL
VAR_INPUT
END_VAR
This^.M_HVE(This^.bWasOn);
M_Recover := bWasOn;
IF (bWasOn) THEN fbLogger(sMsg:='Auto Recovery Initiated.', eSevr:=TcEventSeverity.Info); END_IF;
END_METHOD

METHOD M_SetBits : BOOL
VAR_INPUT
    TermBits : UINT; // The terminal's maximum value in bits
END_VAR
This^.iTermBits := TermBits;
END_METHOD

END_FUNCTION_BLOCK

// ---- POUs/Functions/Gauges/FB_GaugeBase.TcPOU
{attribute 'reflection'}
FUNCTION_BLOCK FB_GaugeBase
VAR
    //Logging
    fbLogger : FB_LogMessage := (eSubsystem:=E_SubSystem.VACUUM);
    ePrevState : E_PressureState;
    tErrorPresent : R_TRIG;
    tAction : R_TRIG; // Primary action of this device (OPN_DO, etc.)
    tOverrideActivated : R_TRIG;
     tState : R_TRIG;
    {attribute 'instance-path'}
    {attribute 'noinit'}
    sPath: STRING;
    // For Persistent Data
    bRestorePersistentData	:	BOOL:=TRUE;
    stateTimer:TON;
    fbGetCurTaskIdx  : GETCURTASKINDEX;
    fbWritePersistentData           : WritePersistentData;
    tRecover: TON;
END_VAR
VAR PERSISTENT
    rVAC_SP	:	REAL;
    rPRO_SP	:	REAL;
    rHYS_PR: REAL;
END_VAR

END_FUNCTION_BLOCK

// ---- UnitTests/Functions/V_TO_INT.TcPOU
{attribute 'no_check'}
FUNCTION V_TO_INT : INT
VAR_INPUT
    analog : REAL;
END_VAR
VAR
    iBits :INT := 30518;
    iFullRange:INT := 10;
END_VAR

if ( iFullRange = 0 ) THEN iFullRange := 10;END_IF
V_TO_INT := REAL_TO_INT(analog * 30518 /iFullRange);

END_FUNCTION

// ---- POUs/ADS/FB_ADS.TcPOU
FUNCTION_BLOCK FB_ADS
VAR_INPUT
END_VAR
VAR_OUTPUT
END_VAR
VAR
     fbLogger : FB_LogMessage := (eSubsystem:=E_SubSystem.FIELDBUS);
    tErrorPresent : R_TRIG;
END_VAR

END_FUNCTION_BLOCK

// ---- POUs/ADS/FB_ADS_WATCHDOG.TcPOU
(*This function block is to be used whenever deivce data going to be read over ADS*)
(*The remote plc has to instantiate this function block in order to write a watchdog variable*)
(*that the ADS read function expects to keep checking*)
FUNCTION_BLOCK FB_ADS_WATCHDOG
VAR_INPUT
    sNetId : String; //NetID of the Destination PLC controller
    nPort : uint; // port number
    sVarName : string;// the variable name of the watchdog on the remote plc.
END_VAR
VAR_OUTPUT
    bError:BOOL;
END_VAR
VAR

    fb_WriteWatchdog:FB_WriteWatchdog;
    ftReset_Watchdog: F_TRIG;
    xFirstPass: BOOL:= true;

END_VAR



ftReset_Watchdog(CLK:= fb_WriteWatchdog.bBusy OR xFirstPass);
xFirstPass := false;

(*calling ADS Watchdog function*)
fb_WriteWatchdog(
    bEnable:= TRUE ,
    sNetId:= sNetId,
    nPort:= nPort,
    nIdxGrp:= ,
    nIdxOffs:= ,
    sVarName:= sVarName,
    tWatchdogTime:= t#30ms,
    bSendNow:= ftReset_Watchdog.Q ,
    bBusy=> ,
    nLastCnt=>  ,
    bError=> bError,
    nErrorId=> );


(*Error*)

END_FUNCTION_BLOCK

// ---- POUs/ADS/FB_TBOOL_ADS.TcPOU
(* This function block is created for interface a boolean singal between different PLCs*)
(* The variable values are read via ADS using the symbol name*)
FUNCTION_BLOCK FB_TBOOL_ADS Extends FB_ADS
VAR_INPUT
    sNetId : String; //NetID of the Destination PLC controller
    nPort : uint; // port number
    sVarName : string;// the variable name of the declared pip/pin function block.
    iWatchdog:UDINT;//The watchdog variable name written to by the remote plc
END_VAR
VAR_OUTPUT
    {attribute 'pytmc' := 'pv: value'}
    bBool : BOOL;
    {attribute 'pytmc' := 'pv: error'}
    bError: BOOL;
END_VAR
VAR
    fb_CheckWatchdog: FB_CheckWatchdog;
    fb_Read: FB_ReadAdsSymByName;
    ftReset: F_TRIG;
    xFirstPass: BOOL:= true;

END_VAR


ftReset(CLK:= fb_Read.bBusy OR xFirstPass);
xFirstPass := false;
(*calling ADS read function*)

fb_Read(
    bRead:=ftReset.Q ,
    sNetId:= sNetId,
    nPort:= nPort,
    sVarName:= sVarName,
    nDestAddr:= ADR(bBool),
    nLen:= SIZEOF(bBool),
    tTimeout:= ,
    eComMode:=eAdsComModeFastCom ,
    bBusy=> ,
    bError=> ,
    nErrorId=> );


(*Error*)
fb_CheckWatchdog(
    bEnable:= TRUE,
    tWatchdogTime:= T#900ms,
    nCnt:= iWatchdog ,
    bWatchdog=> ,
    nLastCnt=> );

bError:= fb_Read.bError OR fb_CheckWatchdog.bWatchdog;
tErrorPresent(CLK:=bError);

IF (fb_Read.bError OR fb_CheckWatchdog.bWatchdog) THEN
    bBool := FALSE; // If there is an error in connection the signal turns to FALSE
END_IF;

(*Logger*)
ACT_Logger();

ACTION ACT_Logger:
IF tErrorPresent.Q THEN
 IF(fb_Read.bError) THEN fbLogger(sMsg:='ADS Read Error', eSevr:=TcEventSeverity.Critical); END_IF;
 IF(fb_CheckWatchdog.bWatchdog) THEN fbLogger(sMsg:='ADS Watchdog Error', eSevr:=TcEventSeverity.Critical); END_IF;
END_IF
END_ACTION

END_FUNCTION_BLOCK

// ---- POUs/Functions/Deprecated/Gauges/FB_MKS317A.TcPOU
(*Deprecated*)
(* This function is for the Pirani MKS 317 connected to a 937A*)
(* This function block is used to provide protection and automatic turn on of ion gauges,
 it also manages the turn on of the AT_VAC boolean, and checks to make sure the pressure is good *)
{attribute 'obsolete' := 'FB_MKS317A has been deprecated and is not valid!'}
FUNCTION_BLOCK FB_MKS317A  Extends FB_GaugeBase
VAR_IN_OUT

END_VAR
VAR_INPUT

END_VAR
VAR_OUTPUT
    {attribute 'pytmc' := '
    pv:
    '}
    PG : ST_VG;
END_VAR
VAR
    rV	:	REAL;
    rMinPressure: REAL := 1E-3;
    rDefaultVAC_SP: REAL :=5E-2; // Default 50 mT
    rValidLoBoundary	:	REAL := 0.2;//Manual page 61
    rValidHiBoundary	:	REAL := 9.7; //manual oage 61
    rDisconnectedBoundary	:	REAL := 0.17;
    rNoSensorBoundary	:	REAL := 10;
    (*IO*)
    i_iPRESS_R AT%I* :INT; // input Pressure // Link to analog Input
END_VAR

(* 937B Logarithmic Output Conversion *)
(* 5-20-2016, Alex Wallace and Scott Stubbs *)
(* 09-28-2018, Margaret Ghaly *)
(* This function will read the pressure from any gauge on a 937A. *)

rV := 10*INT_TO_REAL(PG.i_iPRESS_R)/32767;
PG.rPRESS := LREAL_TO_REAL(EXPT(10,((rV)/0.6)-12)); //manual page 61 937A


//Default setpoint
IF PG.rVAC_SP = 0 THEN
    PG.rVAC_SP := rDefaultVAC_SP;
END_IF

IF (rV <=9.7 ) AND (rV>=0.6) THEN
    PG.eState := Valid; // normal
ELSIF rV >= 0.18 AND rV <= 0.22 THEN
    PG.eState := ValidLo; //LO
    PG.rPRESS := rMinPressure;
ELSIF rV > 9.7 AND rV<= 9.9 THEN
    PG.eState := ValidHi; //HIGH
ELSIF rV < 0.18 THEN
    PG.eState := GaugeDisconnected; //not on
    PG.rPRESS := -1;
ELSE
    PG.eState := PressInvalid; //other fault - could be no gauge, controller powering up etc
    PG.rPRESS := -1;
END_IF

(* Pressure OK check *)
(* Pressure gauge OK checks *)
PG.xPRESS_OK := (rV <=rValidHiBoundary ) AND (rV>=rDisconnectedBoundary);
//PG.xPRESS_OK := (PG.rPRESS >= rMinPressure);

(* Setpoint evaluation *)
PG.xAT_VAC := (*(PG.eState =Valid)*) PG.xPRESS_OK AND PG.rPRESS <= PG.rVAC_SP;

(*Logger*)
ACT_Logger();
(*soft io*)
IO();

ACTION ACT_Logger:
IF (PG.xLog) THEN
//STATE Logger
IF ePrevState <> PG.eState THEN
      CASE PG.eState OF
        ValidHi:
            fbLogger(sMsg:='Gauge pressure valid high.', eSevr:=TcEventSeverity.Info);
        ValidLo:
            fbLogger(sMsg:='Gauge pressure valid low.', eSevr:=TcEventSeverity.Info);
        Valid:
            fbLogger(sMsg:='Gauge pressure valid.', eSevr:=TcEventSeverity.Info);
          GaugeDisconnected:
            fbLogger(sMsg:='Gauge Disconnected.', eSevr:=TcEventSeverity.Critical);
        PressInvalid:
            fbLogger(sMsg:='Gauge pressure invalid.', eSevr:=TcEventSeverity.Warning);
        OoR:
            fbLogger(sMsg:='Gauge pressure out of range.', eSevr:=TcEventSeverity.Warning);
        Starting:
            fbLogger(sMsg:='Gauge starting.', eSevr:=TcEventSeverity.Info);
      END_CASE
      ePrevState := PG.eState;
  END_IF
 END_IF
END_ACTION

ACTION IO:
PG.i_iPRESS_R :=i_iPRESS_R;
PG.sPath := sPath;
END_ACTION

END_FUNCTION_BLOCK

// ---- POUs/Functions/Deprecated/Gauges/FB_MKS500_EP.TcPOU
(*Deprecated*)
(* This function is for the Cold Cathode MKS 500 connected to Beckhoff EP boxes.
A separate function block is necessary for the MKS500-to-EP box interface beacuse the EP
boxes do not natively support the 5v IO signals on the MKS500 gauge.*)
(*This function provides ILK and Set Point Protection for the Cold Cathode*)
(* 500 Logarithmic Output Conversion, factory default configuration *)
{attribute 'obsolete' := 'FB_MKS500_EP has been deprecated and is not valid!'}
FUNCTION_BLOCK FB_MKS500_EP EXTENDS FB_GaugeBase
VAR_IN_OUT

END_VAR
VAR_INPUT

    PG	:	ST_VG;
END_VAR
VAR_OUTPUT
{attribute 'pytmc' := '
    pv:
    '}
    IG : ST_VG;
END_VAR
VAR
    rV : REAL;
    GaugeTurnOnTmr : TON;

    (*IOs to be linked*)
    /// Controls and I/Os
    i_iPRESS_R AT %I* :INT; // input Pressure // Link to analog Input
    q_xHV_DIS AT %Q* : BOOL; // Enable High Voltage when True // 'TcLinkTo' (EP2624) ^Output
    //
END_VAR

VAR CONSTANT
    // Ranges has to match the configurator software
    pBase : REAL :=1.0E-10;//default curve base pressure is 1E-10. Confusing since can't actually read that low using analog out.
    vBase : REAL := 1;
    vDisconnected : REAL:= 0.5;
    vSlope : REAL := 1.0;
    vGaugeOff: REAL := 9.8;
    vNoDischarge: REAL := 9.3;
    MinPressure: REAL := 1E-10;
    cDefaultPressure : REAL := 0;
END_VAR

(* 500 Logarithmic Output Conversion, factory default configuration *)
{attribute 'obsolete' := 'FB_VCC_NO has been deprecated and is not valid!'}
rV := 10*INT_TO_REAL(IG.i_iPRESS_R)/32767;

(* Set Guage State based on the Analog voltage*)
IF rV < vDisconnected THEN
    IG.eState := GaugeDisconnected;
    IG.rPRESS := cDefaultPressure;
ELSIF rV >= vDisconnected AND rV < (vNoDischarge -0.3)  THEN
    IG.eState := Valid;
    IG.rPRESS := LREAL_TO_REAL(EXPT(10,((rV-vBase)/vSlope+LOG(pBase))));
ELSIF rV >= (vNoDischarge -0.3) AND rV <(vGaugeOff -0.3)   THEN
    IG.eState := Starting;
    IG.rPRESS := LREAL_TO_REAL(EXPT(10,((rV-vBase)/vSlope+LOG(pBase))));
ELSIF rV >= (vGaugeOff -0.3) THEN
    IG.eState := Off;
    IG.rPRESS := LREAL_TO_REAL(EXPT(10,((rV-vBase)/vSlope+LOG(pBase))));
ELSE
    IG.eState := OoR;
    IG.rPRESS := LREAL_TO_REAL(EXPT(10,((rV-vBase)/vSlope+LOG(pBase))));
END_IF


(* Ion Gauge Protection Functions *)
(* If the PG pressure is greater than the VG.PRO_SP then the gauge is disabled *)
(* If the PG pressure is less than the VG.PRO_SP then the gauge is enabled *)
(* This FB also implements some hysteresis so the gauge doesn't have rapid power cycling while near the turn on boundary *)


IF PG.rPRESS <= IG.rPRO_SP AND PG.xPRESS_OK THEN

    IG.q_xHV_DIS := IG.xHV_SW;
    IG.xILKOk := TRUE;
ELSIF IG.q_xHV_DIS THEN
    IF IG.rPRESS > (IG.rPRO_SP + IG.rHYS_PR)  OR PG.rPRESS > (IG.rPRO_SP + IG.rHYS_PR) THEN
        IG.q_xHV_DIS := FALSE;
        IG.xHV_SW := FALSE;
    END_IF
ELSE
    IG.q_xHV_DIS := FALSE;
    IG.xHV_SW := FALSE;
    IG.xILKOk := FALSE;
END_IF

(* Pressure gauge OK checks *)

GaugeTurnOnTmr(IN:=IG.q_xHV_DIS, PT:=T#10S, Q=>IG.xTurnOnTime);


//Backwards compatibility
IG.xPRESS_OK := (IG.eState = Valid) OR IG.xBAKEOUT;

(* Setpoint evaluation *)
IG.xAT_VAC := (IG.xPRESS_OK AND (IG.rPRESS < IG.rVAC_SP)) OR IG.xBAKEOUT AND (IG.eState = Valid) ;

ACT_Logger();
(*Soft IO Linking*)
// check ethercat Diagnostics
IO();

ACTION ACT_Logger:
IF (IG.xLog) THEN
// ILK logger
IF NOT IG.xILKOk AND NOT IG.q_xHV_DIS THEN
         fbLogger(sMsg:='Lost external interlock while gauge was on.', eSevr:=TcEventSeverity.Critical);
END_IF


// Log Action
tAction(CLK:=  IG.q_xHV_DIS);
IF tAction.Q THEN fbLogger(sMsg:='Ion gauge commanded to switch on', eSevr:=TcEventSeverity.Info); END_IF



//STATE Logger
IF ePrevState <> IG.eState THEN
      CASE IG.eState OF
        ValidHi:
            fbLogger(sMsg:='Gauge pressure valid high.', eSevr:=TcEventSeverity.Info);
        ValidLo:
            fbLogger(sMsg:='Gauge pressure valid low.', eSevr:=TcEventSeverity.Info);
        Valid:
            fbLogger(sMsg:='Gauge pressure valid.', eSevr:=TcEventSeverity.Info);
          GaugeDisconnected:
            fbLogger(sMsg:='Gauge Disconnected.', eSevr:=TcEventSeverity.Critical);
        PressInvalid:
            fbLogger(sMsg:='Gauge pressure invalid.', eSevr:=TcEventSeverity.Warning);
        OoR:
            fbLogger(sMsg:='Gauge pressure out of range.', eSevr:=TcEventSeverity.Warning);
        Starting:
            fbLogger(sMsg:='Gauge starting.', eSevr:=TcEventSeverity.Info);
      END_CASE
      ePrevState := IG.eState;
  END_IF
END_IF
END_ACTION

ACTION IO:
(*soft link inputs*)
IG.i_iPRESS_R:=	i_iPRESS_R;
(*soft link outputs*)
q_xHV_DIS := IG.q_xHV_DIS;

IG.sPath := sPath;
END_ACTION

METHOD M_HVE : BOOL
VAR_INPUT
        enable:bool; // set to true to enable, false to disable;
END_VAR

this^.IG.xHV_SW:= NOT(enable);
END_METHOD

END_FUNCTION_BLOCK

// ---- POUs/Functions/Deprecated/Valves/FB_VCC_NO.TcPOU
(*Deprecated*)
(* This Function Block Implements Basic Functionality for NO Vent Valves VVC *)
(* Note Interlock Logic is External *)
{attribute 'obsolete' := 'FB_VCC_NO has been deprecated and is not valid!'}
FUNCTION_BLOCK FB_VCC_NO
VAR_IN_OUT
    {attribute 'pytmc' := 'pv:'}
    iq_stValve : ST_VCC_NO;

END_VAR
VAR_INPUT
    i_xExtILK_OK:BOOL; (*Other External Interlock, Set to True when no external interlock is required*)
    i_xOverrideMode : BOOL; (*To be linked to global override bit. This Overrides Vacuum logic only, EPS, MPS and PMPS are still enforces*)

END_VAR
VAR_OUTPUT
END_VAR
VAR

    tonOvrd	:	TON;
    tonDelOK : TON;
    rtOK	:	R_TRIG;
    (*IO*)
    xCLS_DO	AT%Q*: BOOL;

END_VAR


IF NOT iq_stValve.xCLS_OK THEN
iq_stValve.pv_xCLS_SW := FALSE;
END_IF

(* Override logic *)
(* Goal: give ability to override, but do so in a way that people won't forget it.
Solution: Override only after ten seconds of override, protect against blips,
when the valve permission goes true for more than ten seconds consistently, remove override
*)

tonDelOK(IN:=iq_stValve.xCLS_OK, PT:=T#10S);
rtOK(CLK:=tonDelOK.Q);
IF rtOK.Q THEN iq_stValve.pv_xOvrdCls :=FALSE; END_IF

//Override timer
tonOvrd(IN:=iq_stValve.pv_xOvrdCls, PT:=T#10S);

(* Here's where the valve is closed *)
iq_stValve.xCLS_DO := (iq_stValve.pv_xCLS_SW AND iq_stValve.xCLS_OK) OR (tonOvrd.Q AND i_xOverrideMode);

ACTION ACT_IO:
(*inputs*)
iq_stValve.xOverrideMode := i_xOverrideMode;
(*outputs*)
xCLS_DO:= iq_stValve.xCLS_DO;
END_ACTION

METHOD M_Close : BOOL
VAR_INPUT
        close:BOOL; //True to CLose, False to OPEN
END_VAR
// Checking the VAR_IN_OUT reference, leave the current method in case of invalid reference
IF NOT __ISVALIDREF(iq_stValve) THEN
    RETURN;
END_IF

THIS^.iq_stValve.pv_xCLS_SW :=Close;
END_METHOD

END_FUNCTION_BLOCK

// ---- POUs/Functions/Deprecated/Gauges/FB_PressureState.TcPOU
(*Deprecated*)
FUNCTION_BLOCK FB_PressureState
VAR_INPUT
    i_rV	:	REAL;
    i_rVMin	:	REAL := 0.01; // Anything less than this voltage is considered disconnected
    i_rVMax :	REAL := 10.5; // Anything more than this is considered invalid
    i_IGTurnOnTime	:	TIME := T#10S;

    i_MinPressure	:	REAL;
    i_MaxPressure	:	REAL;
END_VAR
VAR_OUTPUT
    q_eState 	:	E_PressureState;
END_VAR
VAR_IN_OUT
    iq_stVG	:	ST_VG;
END_VAR
VAR
    tonGaugeTurnOnTmr : TON;
END_VAR

(* Pressure State Evaluation
A. Wallace, 2016-8-31

This FB serves to evaluate the state of the pressure based on the raw voltage, pressure, and gauge state.

*)
// Is the gauge plugged in, and within a reasonable range?
IF i_rV < i_rVMin THEN
    q_eState := GaugeDisconnected;
ELSIF i_rV > i_rVMax THEN
    q_eState := PressInvalid;
ELSE
    // Is the gauge reading back a pressure that makes sense?
    CASE iq_stVG.eTYPE OF
        IG903:
            tonGaugeTurnOnTmr(IN:=iq_stVG.q_xHV_DIS, PT:=i_IGTurnOnTime, Q=>iq_stVG.xTurnOnTime);
            IF iq_stVG.q_xHV_DIS THEN
                IF tonGaugeTurnOnTmr.Q THEN
                    IF iq_stVG.rPRESS >= i_MinPressure AND iq_stVG.rPRESS <= i_MaxPressure THEN
                        q_eState := Valid;
                    ELSE
                        q_eState := OoR;
                    END_IF
                ELSE
                        q_eState := Starting;
                END_IF
            ELSE
                q_eState := Off;
            END_IF
        IG909:
            IF iq_stVG.q_xHV_DIS THEN
                IF iq_stVG.rPRESS >= i_MinPressure AND iq_stVG.rPRESS <= i_MaxPressure THEN
                    q_eState := Valid;
                ELSE
                    q_eState := OoR;
                END_IF
            ELSE
                q_eState := Off;
            END_IF
        PG907, PG925, PG722B:
            IF iq_stVG.rPRESS >= i_MinPressure AND iq_stVG.rPRESS <= i_MaxPressure THEN
                q_eState := Valid;
            ELSIF iq_stVG.rPRESS < i_MinPressure THEN
                q_eState := ValidLo;
            ELSE
                q_eState := ValidHi;
            END_IF
        ELSE
            q_eState := PressInvalid;
    END_CASE
END_IF


iq_stVG.eState := q_eState;

// Legacy Press OK boolean eval
iq_stVG.xPRESS_OK := q_eState >= gc_GaugeValidState;

END_FUNCTION_BLOCK

// ---- POUs/Functions/Deprecated/Valves/FB_VCC.TcPOU
(*Deprecated*)
(* THE FB_VCC FUNCTION BLOCK IS DEPRECATED. USE FB_VVC INSTEAD. *)
(* This Function Block Implements Basic Functionality for Vent Valves VVC *)
(* Note Interlock Logic is External *)
FUNCTION_BLOCK FB_VCC
VAR_IN_OUT

END_VAR
VAR_INPUT
    i_xExtILK_OK:BOOL; (*Other External Interlock, Set to True when no external interlock is required*)
    i_xOverrideMode : BOOL; (*To be linked to global override bit. This Overrides Vacuum logic only*)
END_VAR
VAR_OUTPUT
    {attribute 'pytmc' := '
    pv:
    '}
    iq_stValve : ST_VVC;
END_VAR
VAR

    tonOvrd	:	TON;
    tonDelOK : TON;
    rtOK	:	R_TRIG;

    (*IO*)
    q_xOPN_DO	AT%Q*: BOOL;

END_VAR


iq_stValve.xOPN_OK := i_xExtILK_OK;

IF NOT iq_stValve.xOPN_OK THEN
iq_stValve.pv_xOPN_SW := FALSE;
END_IF

(* Override logic *)
(* Goal: give ability to override, but do so in a way that people won't forget it.
Solution: Override only after ten seconds of override, protect against blips,
when the valve permission goes true for more than ten seconds consistently, remove override
*)

tonDelOK(IN:=iq_stValve.xOPN_OK, PT:=T#10S);
rtOK(CLK:=tonDelOK.Q);
IF rtOK.Q THEN iq_stValve.xOvrdOpn :=FALSE; END_IF

//Override timer
tonOvrd(IN:=iq_stValve.xOvrdOpn, PT:=T#10S);

(* Here's where the valve opens *)
iq_stValve.q_xOPN_DO := (iq_stValve.pv_xOPN_SW AND iq_stValve.xOPN_OK) OR (tonOvrd.Q AND i_xOverrideMode);

(*IO Mapping*)
ACT_IO();

ACTION ACT_IO:
(*inputs*)
iq_stValve.xOverrideMode := i_xOverrideMode;
(*outputs*)
q_xOPN_DO:= iq_stValve.q_xOPN_DO;
END_ACTION

METHOD PUBLIC M_IsClosed : BOOL
VAR_INPUT
END_VAR
M_IsClosed := NOT This^.q_xOPN_DO;
END_METHOD

METHOD PUBLIC M_IsOpen : BOOL
VAR_INPUT
END_VAR
M_IsOpen := This^.q_xOPN_DO;
END_METHOD

// Use this Methode to Open or close the valve by setting the OPN_SW to the input value.
METHOD PUBLIC M_Set_OPN_SW : BOOL
VAR_INPUT
        value:BOOL;  //True to SET, False to RESET
END_VAR
This^.iq_stValve.pv_xOPN_SW := value;
END_METHOD

END_FUNCTION_BLOCK

// ---- POUs/Functions/Deprecated/Valves/FB_VGC_AP.TcPOU
(*Deprectated*)
(* This function block implements basic functionality for Isolation Gate Valves with Appertures*)
(* This function block interlock is as follows:
1. The valve can be opened when the difference between the pressures on both sides is
less than the maximum differential pressure.
2. This rule persists until the pressures on both sides are lower than the vacuum-setpoint.
3. Once at-vac, the valve will close if the pressure on either side rises above the setpoint.*)
(*This function block also implements PMPS and EPS interlocks, as well as Fast MPS trigger*)
(* MPS is triggered differently than the VGC *)
{attribute 'no_check'}
{attribute 'obsolete' := 'FB_VGC_AP has been deprecated and is not valid!'}
FUNCTION_BLOCK FB_VGC_AP
VAR_IN_OUT

END_VAR
VAR_INPUT
    (*Upstream Gauge, usually ion gauge*)
    i_stUSG	:	ST_VG;
    (*Downstream Gauge, usually ion gauge*)
    i_stDSG	:	ST_VG;
    {attribute 'pytmc' := '
    pv: Dis_DPIlk
    '}
    i_xDis_DPIlk : BOOL := FALSE;  (* Set to true when calling the function to disable the differential pressure interlock *)
    {attribute 'pytmc' := '
    pv: EPS_OK
    '}
    i_xEPS_OK:	BOOL	:= TRUE; (*External EPS interlock, Set to TRUE when no EPS interlock is required, otherwise set to correct interlock signal*)
    {attribute 'pytmc' := '
    pv: MPS_OK
    '}
    i_xPMPS_OK:	BOOL	; (*External MPS interlock, Set to TRUE when no PMPS interlock is required*)
    i_xExt_OK: BOOL; (*Other External Interlock, Set to True when no external interlock is required. If this Valve is neigboring a Fast Shutter this should be linked to the fast shutter xVAC_FAULT_OK*)
    i_xOverrideMode : BOOL; (*To be linked to global override bit. This Overrides Vacuum logic only, EPS, MPS and PMPS are still enforces*)
    // Reset fault
    {attribute 'pytmc' := '
    pv: FF_Reset
    '}
    i_xReset: BOOL;
    i_sDevName : T_MaxString :=  'VGC'; // Device name for diagnostic
END_VAR
VAR_OUTPUT
    {attribute 'pytmc' := '
    pv:
    '}
    iq_stValve : ST_VGC; (* All valve data and states will be in this struct*)

    {attribute 'pytmc' := '
    pv: MPS_FAULT_OK
    '}
    xMPS_OK:	BOOL; (*MPS Fast OK, is set when the Valve is Open*)
END_VAR
VAR_IN_OUT
    io_fbFFHWO    :    FB_HardwareFFOutput;
END_VAR
VAR
    // PMPS
    fbFF    :    FB_FastFault :=(
        i_DevName := 'VGC Aptr',
        i_Desc := 'Fault occurs when the valve is not in open state',
        i_TypeCode := 16#1010);
    //g_FastFaultOutput1	:	FB_HardwareFFOutput;

    {attribute 'instance-path'}
    {attribute 'noinit'}
    sPath: STRING;

    rDiffPressAllowed	:	REAL := 22.5; // Torr, Default value comes from Vat Valve Manual
    rDiffPress : REAL;
    set : BOOL;
    reset: BOOL;

    xFirstPass	:	BOOL;
    fbFSInit		:	R_TRIG;

    tonDelOK : TON;
    rtOK	:	R_TRIG;
    tonOvrd	:	TON;

    tDelOK	:	TIME := T#60S;
    tOvrd	:	TIME := T#10s;


    (* Timeouts*)
    tTimeOutDuration: TIME:= T#30S;
    tOPNtimeout: TON;
    tCLStimeout:TON;

     // For logging
    fbLogger : FB_LogMessage := (eSubsystem:=E_SubSystem.VACUUM);
    ePrevState : E_VGC;
    tErrorPresent : R_TRIG;
    tAction : R_TRIG; // Primary action of this device (OPN_DO, PUMP_RUN, etc.)
    tOverrideActivated : R_TRIG;



    (*IO*)
    i_xOpnLS	AT%I*: BOOL;
    i_xClsLS	AT%I*: BOOL;
    q_xOPN_DO	AT%Q*: BOOL;

END_VAR

(* Vacuum gate valve
A. Wallace
16-10-29

A gate valve isolates vacuum volumes. Ideally it can be opened when a system is vented
to allow for faster pumping, and will close when high vacuum is lost.

The following behavior is good for valves in something like a gas attenuator.
This function block does the following:
1. The valve can be opened when the difference between the pressures on both sides is
less than the maximum differential pressure.
2. This rule persists until the pressures on both sides are lower than the vacuum-setpoint.
3. Once at-vac, the valve will close if the pressure on either side rises above the setpoint.

Alternatively, the differential pressure interlock can be disabled so the valve may only be opened
if the pressure on both sides is lower than the at-vacuum-setpoint. You want this behavior if
the valve is to be used in a UHV section.

Hysteresis is employed to ensure a smooth transition from vented/pumping down, to at-vac.

Finally, an override system is built in so you can bypass all the interlocking logic and
get back online.
*)
(* 10/1/2018 Margaret Ghaly included EPS, PMPS Checkes and MPS trigger signals*)


fbFSInit( CLK := TRUE, Q => xFirstPass);
(*IO Mapping*)
ACT_IO();

(* On first PLC pass, put valve into vented state, which implies a closed valve *)
IF xFirstPass THEN
    iq_stValve.eVGC_State := Vented;
    iq_stValve.pv_xOPN_SW := FALSE;
    fbFF.i_DevName := i_sDevName;
END_IF


